// ---- Templates/GVLs/DPAD/Labels/Composition/LblCmpAC.TcGVL
{region '#Template'}
	{attribute 'Version' := '0.0.1.0'}
	{attribute 'Tags' := '"LCID": "1031", "Text": "GVL, AC, DPAD, Plants, ObjectName, Description"'}
	{attribute 'Tags' := '"LCID": "1033", "Text": "GVL, AC, DPAD, Plants, ObjectName, Description"'}
	{attribute 'Description' := '"LCID": "1031", "Text": "AC Labels Kompensation"'}
	{attribute 'Description' := '"LCID": "1033", "Text": "AC labels compensation"'}
{endregion}

{attribute 'qualified_only'}
VAR_GLOBAL
///////////////////////
//	Aggregates\Cooler	
	Cooler_TFl							:FB_BA_Label	:= LblAggregates.TemperatureFlow;	
	Cooler_TRt							:FB_BA_Label	:= LblAggregates.TemperatureReturnFlow;	

	Cooler_HSuACtrl_Ctrl				:FB_BA_Label	:= LblFunctions.LoopObject; 
	Cooler_HSuACtrl_Dehumf				:FB_BA_Label	:= LblControl.OperationalMessageDehumidification;	

	Cooler_TSuACtrl						:FB_BA_Label	:= LblControl.SupplyAirTemperatureControl;
	Cooler_TSuACtrl_Ctrl				:FB_BA_Label	:= LblFunctions.LoopObject; 

	Cooler_Vlv							:FB_BA_Label	:= LblAggregates.Valve;
	Cooler_Pu							:FB_BA_Label	:= LblAggregates.Pump;

//	Aggregates\ERC
	ERC_DiffPrssSwi						:FB_BA_Label	:= LblAggregates.PressureDifferential;												 										 
	ERC_IcePrtcRamp						:FB_BA_Label	:= LblControl.EnergyRecoveryDeicingRamp;
	ERC_Motor							:FB_BA_Label	:= LblAggregates.HeatRecovery;
	ERC_TExhACtrl						:FB_BA_Label	:= LblControl.ExhaustAirTemperatureControl;
	ERC_TSuACtrl						:FB_BA_Label	:= LblControl.SupplyAirTemperatureControl;
	ERC_TSuACtrl_Ctrl					:FB_BA_Label	:= LblFunctions.LoopObject; 

	ERC_DiffPrssSensor					:FB_BA_Label	:= LblAggregates.PressureDifferential;	
	ERC_Damping							:FB_BA_Label	:= LblAggregates.PressureDifferential;
	ERC_IcePrtcDiffPrssCtrl				:FB_BA_Label	:= LblControl.ExhaustAirTemperatureControl;
	ERC_Dmp								:FB_BA_Label	:= LblAggregates.VentilationDamperSupplyAir;	
	ERC_ByDmp							:FB_BA_Label	:= LblAggregates.VentilationDamperBypassAir;

//	Aggregates\Humidifier
	Humf_SuACtrl_Ctrl					:FB_BA_Label	:= LblFunctions.LoopObject; 
		
//	Aggregates\MixedAir
	Mix_TSuACtrl						:FB_BA_Label	:= LblControl.SupplyAirTemperatureControl;
	Mix_TSuACtrl_Ctrl					:FB_BA_Label	:= LblFunctions.LoopObject; 
	Mix_StartUpRamp						:FB_BA_Label	:= LblControl.MixedAirStartUpRamp;
	Mix_DmpMixA							:FB_BA_Label	:= LblAggregates.VentilationDamperMixAir;	
	Mix_DmpOuA							:FB_BA_Label	:= LblAggregates.VentilationDamperOutsideAir;	
	Mix_DmpExhA							:FB_BA_Label	:= LblAggregates.VentilationDamperExhaustAir;	

//	Aggregates\pre-heater
	PreHtr_TFl							:FB_BA_Label	:= LblAggregates.TemperatureFlow;	
	PreHtr_TRt							:FB_BA_Label	:= LblAggregates.TemperatureReturnFlow;	
	PreHtr_TSuACtrl						:FB_BA_Label	:= LblControl.SupplyAirTemperatureControl;
	PreHtr_TSuACtrl_Ctrl				:FB_BA_Label	:= LblFunctions.LoopObject; 
	PreHtr_TFrost						:FB_BA_Label	:= LblControl.TemperatureFrost;	
	PreHtr_TFrostPrtcCtrlAir			:FB_BA_Label	:= LblControl.FrostProtectionControl;
	PreHtr_FrostThermostat				:FB_BA_Label	:= LblAggregates.FrostProtectionMonitor;												 										 
	PreHtr_FrostThermostat_Input		:FB_BA_Label	:= LblFunctions.DangerAlarm;
	PreHtr_Vlv							:FB_BA_Label	:= LblAggregates.Valve;
	PreHtr_Pu							:FB_BA_Label	:= LblAggregates.Pump;		
	PreHtr_TRtCtrl						:FB_BA_Label	:= LblControl.ReturnWaterControl;
	PreHtr_TRtCtrl_SpTRtW				:FB_BA_Label	:= LblFunctions.Setpoint;
	PreHtr_TRtCtrl_PreRinseDelay		:FB_BA_Label	:= LblControl.DelayOn;
	PreHtr_TRtCtrl_PreRinseDelay_TiDly	:FB_BA_Label	:= LblControl.PreRinseDuration;
	PreHtr_TRtCtrl_PreRinseDst			:FB_BA_Label	:= LblControl.DisturbancePreRinse;	 								 
	PreHtr_TRtCtrl_PreRinseSp			:FB_BA_Label	:= LblControl.CalculationPreRinseSetpoint;			
	PreHtr_TRtCtrl_Ctrl					:FB_BA_Label	:= LblFunctions.LoopObject; 		
	
	PreHtr_ProcessPreRinse				:FB_BA_LabelProcess	:= LblControl.ProcPreRinse;

//	Aggregates\re-heater
	ReHtr_TFl							:FB_BA_Label	:= LblAggregates.TemperatureFlow;	
	ReHtr_TRt							:FB_BA_Label	:= LblAggregates.TemperatureReturnFlow;	
	ReHtr_TSuACtrl						:FB_BA_Label	:= LblControl.SupplyAirTemperatureControl;
	ReHtr_TSuACtrl_Ctrl					:FB_BA_Label	:= LblFunctions.LoopObject; 
	ReHtr_Vlv							:FB_BA_Label	:= LblAggregates.Valve;
	ReHtr_Pu							:FB_BA_Label	:= LblAggregates.Pump;		
		
///////////////////////
//	General
	General_OpModMan					:FB_BA_Label	:= LblControl.OperationModeSelection;							
	General_Sched						:FB_BA_Label	:= LblFunctions.Scheduler;							
	General_OpModPr						:FB_BA_Label	:= LblControl.PresentOperationMode;		
	
//	Summer night cooling
	General_SumNgtCol_WthTLoLmt			:FB_BA_Label	:= LblControl.OutsideTemperatureLowLimit;			
	General_SumNgtCol_RmTHys			:FB_BA_Label	:= LblControl.HysteresisRoomTemperature;			
	General_SumNgtCol_SwiOnDiffT		:FB_BA_Label	:= LblControl.OnValueDifferenceOutsideInsightTemperature;			
	General_SumNgtCol_SwiOffDiffT		:FB_BA_Label	:= LblControl.OffValueDifferenceOutsideInsightTemperature;			
	General_SumNgtCol_Q					:FB_BA_Label	:= LblFunctions.OperationalMessage;												 
	General_SumNgtCol_Sched				:FB_BA_Label	:= LblFunctions.Scheduler;		
///////////////////////
//	Setpoint\Temperature
	SpTRm_X1							:FB_BA_Label	:= LblControl.X01;	
	SpTRm_X2							:FB_BA_Label	:= LblControl.X02;	
	SpTRm_X3							:FB_BA_Label	:= LblControl.X03;	
	SpTRm_X4							:FB_BA_Label	:= LblControl.X04;	
	
	SpTRm_Y1							:FB_BA_Label	:= LblControl.Y01;
	SpTRm_Y2_3							:FB_BA_Label	:= LblControl.Y02_03;
	SpTRm_Y4							:FB_BA_Label	:= LblControl.Y03;
	SpTRm_Sp							:FB_BA_Label	:= LblFunctions.SetpointCalculated;
	
	SpTRm_SpColX1						:FB_BA_Label	:= LblControl.SummerCompensationX1;	
	SpTRm_SpColX2						:FB_BA_Label	:= LblControl.SummerCompensationX2;	
	SpTRm_SpColY1						:FB_BA_Label	:= LblControl.SummerCompensationY1;	
	SpTRm_SpColY2						:FB_BA_Label	:= LblControl.SummerCompensationY2;	
	SpTRm_SpColYMin						:FB_BA_Label	:= LblControl.SummerCompensationYmin;
	SpTRm_SpColYMax						:FB_BA_Label	:= LblControl.SummerCompensationYmax;	
	SpTRm_SpCol							:FB_BA_Label	:= LblControl.SummerCompensationSp;	
	
	SpTRm_SpHtgX1						:FB_BA_Label	:= LblControl.WinterCompensationX1;	
	SpTRm_SpHtgX2						:FB_BA_Label	:= LblControl.WinterCompensationX2;	
	SpTRm_SpHtgY1						:FB_BA_Label	:= LblControl.WinterCompensationY1;	
	SpTRm_SpHtgY2						:FB_BA_Label	:= LblControl.WinterCompensationY2;	
	SpTRm_SpHtgYMin						:FB_BA_Label	:= LblControl.WinterCompensationYmin;
	SpTRm_SpHtgYMax						:FB_BA_Label	:= LblControl.WinterCompensationYmax;		
	SpTRm_SpHtg							:FB_BA_Label	:= LblControl.WinterCompensationSp;	
	
	SpTSuA_SelSpErc						:FB_BA_Label	:= LblControl.OperationModeSelection;							
	SpTSuA_SpErc						:FB_BA_Label	:= LblFunctions.SetpointCalculated;	

	TCasCtrl_SpHtg						:FB_BA_Label	:= LblControl.SuppyAirTempSetpointHeaterCalc;			
	TCasCtrl_SpCol						:FB_BA_Label	:= LblControl.SuppyAirTempSetpointCoolerCalc;			
	TCasCtrl_SpErc						:FB_BA_Label	:= LblControl.SuppyAirTempSetpointERCCalc;			
	TCasCtrl_Ctrl						:FB_BA_Label	:= LblFunctions.LoopObjectCascadeSupplyAirTemperature; 			
	TCasCtrl_SelSpErc					:FB_BA_Label	:= LblControl.OperationModeSelection;							
//	Setpoint\Humidity
	HumCasCtrl_Ctrl						:FB_BA_Label	:= LblFunctions.LoopObjectCascadeSupplyAirHumidity; 	
	SpHum_SpH							:FB_BA_Label	:= LblControl.SetpointRelHumidity;			
	SpHum_SpX							:FB_BA_Label	:= LblControl.SetpointCalculatedAbsHumidity;
	SpHum_SpHHumf						:FB_BA_Label	:= LblControl.SetpointRelHumidityHumidification;			
	SpHum_SpHDehumf						:FB_BA_Label	:= LblControl.SetpointRelHumidityDehumidification;			
	SpHum_SpXHumf						:FB_BA_Label	:= LblControl.SetpointCalculatedAbsHumidityHumidification;	
	SpHum_SpXDehumf						:FB_BA_Label	:= LblControl.SetpointCalculatedAbsHumidityDehumidification;


//	Sonderlösung - eventuelle Überarbeitung
	PlantControlStatus   	:FB_BA_Label2x :=(iAggregate:=LblControl.PlantControl,		iFunction:=LblFunctions.Status);
	TSequenceControlStatus  :FB_BA_Label2x :=(iAggregate:=LblControl.TSequenceControl,	iFunction:=LblFunctions.Status);		

//	AHU	
	AHU_TOuA						:FB_BA_Label	:= LblAggregates.TemperatureOutside;	
	AHU_TExhA						:FB_BA_Label	:= LblAggregates.TemperatureExhaustAir;	
	AHU_TSuA						:FB_BA_Label	:= LblAggregates.TemperatureSupplyAir;	
	AHU_TExtA						:FB_BA_Label	:= LblAggregates.TemperatureExtractAir;	
	AHU_TRm							:FB_BA_Label	:= LblAggregates.TemperatureRoomAir;	
	AHU_DiffPrssOuAFilt				:FB_BA_Label	:= LblAggregates.PressureDifferentialOutsideAirFilter;	
	AHU_FiltOuAMonit				:FB_BA_Label	:= LblAggregates.AirFilterOutsideAir;
	AHU_DiffPrssExtAFilt			:FB_BA_Label	:= LblAggregates.PressureDifferentialExtractAirFilter;	
	AHU_FiltExtAMonit				:FB_BA_Label	:= LblAggregates.AirFilterExtractAir;
	AHU_SumNgtCol					:FB_BA_Label	:= LblControl.SummerNightCooling;
	AHU_OpMod						:FB_BA_Label	:= LblControl.OperationMode;
	AHU_OuADmp						:FB_BA_Label	:= LblAggregates.VentilationDamperOutsideAir;
	AHU_SuAPrss						:FB_BA_Label	:= LblAggregates.PressureSupplyAir;	
	AHU_SuADiffPrss					:FB_BA_Label	:= LblAggregates.PressureDifferentialSupplyAirFan;	
	AHU_SuAFan						:FB_BA_Label	:= LblAggregates.FanSupplyAir;
	AHU_SuADiffPrssMonit			:FB_BA_Label	:= LblControl.DifferencePressureMonitoringSupplyAirFan;
	AHU_ExhADmp						:FB_BA_Label	:= LblAggregates.VentilationDamperExhaustAir;
	AHU_ExtAPrss					:FB_BA_Label	:= LblAggregates.PressureExtractAir;	
	AHU_ExtADiffPrss				:FB_BA_Label	:= LblAggregates.PressureDifferentialExtractAirFan;	
	AHU_ExtAFan						:FB_BA_Label	:= LblAggregates.FanExtractAir;
	AHU_ExtADiffPrssMonit			:FB_BA_Label	:= LblControl.DifferencePressureMonitoringExtractAirFan;
	AHU_SpTRm						:FB_BA_Label	:= LblControl.SetpointCalculation;
	AHU_TCasCtrl					:FB_BA_Label	:= LblControl.CascadeSupplyAirControl;
	AHU_TSeqLink					:FB_BA_Label2x	:= TSequenceControlStatus;
	AHU_PreHtr						:FB_BA_Label	:= LblControl.PreHeater;
	AHU_Erc							:FB_BA_Label	:= LblControl.EnergyRecovery;
	AHU_Col							:FB_BA_Label	:= LblControl.Cooler;
	AHU_PlantCtrl					:FB_BA_Label2x	:= PlantControlStatus;	



	
END_VAR

// ---- Templates/GVLs/DPAD/Labels/Composition/LblCmpGeneral.TcGVL
{region '#Template'}
	{attribute 'Version' := '0.0.1.0'}
	{attribute 'Tags' := '"LCID": "1031", "Text": "GVL, General, DPAD, Plants, ObjectName, Description"'}
	{attribute 'Tags' := '"LCID": "1033", "Text": "GVL, General, DPAD, Plants, ObjectName, Description"'}
	{attribute 'Description' := '"LCID": "1031", "Text": "Allgemein Labels Kompensation"'}
	{attribute 'Description' := '"LCID": "1033", "Text": "General labels compensation"'}
{endregion}

{attribute 'qualified_only'}
VAR_GLOBAL
	BuildingAlarms_FireAlert						: FB_BA_Label := LblControl.FireAlert;
	BuildingAlarms_Bgly								: FB_BA_Label := LblControl.Burglary;
	BuildingAlarms_CentSwiOff						: FB_BA_Label := LblControl.CentralSwitchOff;
                                  				
	BuildingMode_OpModMan							: FB_BA_Label := LblControl.BuildingModeManual;
	BuildingMode_OpModPr							: FB_BA_Label := LblControl.BuildingModeActual;
	BuildingMode_Sched								: FB_BA_Label := LblControl.BuildingModeSched;
                                  				
	BuildingGlobal_BuildAlm							: FB_BA_Label := LblControl.BuildingAlarms;
	BuildingGlobal_BuildMode						: FB_BA_Label := LblControl.BuildingMode;
	
	ControlCabinet_Fuse								: FB_BA_Label := LblControl.Fuse;	
	ControlCabinet_Fuse_Input						: FB_BA_Label := LblFunctions.Fault;	
	ControlCabinet_LampFault						: FB_BA_Label := LblControl.EventIndicationLamp;			
	ControlCabinet_LampFault_Cmd					: FB_BA_Label := LblFunctions.SwitchingCommand;			
	ControlCabinet_AckButton 						: FB_BA_Label := LblControl.Acknowledge;	
	ControlCabinet_AckButton_Input					: FB_BA_Label := LblControl.ButtonLocalAcknowledgement;
	ControlCabinet_AckButton_Value					: FB_BA_Label := LblControl.ButtonRemoteAcknowledgement;
	ControlCabinet_RstHw							: FB_BA_Label := LblControl.AcknowledgeCommand;			
	ControlCabinet_RstHw_Cmd						: FB_BA_Label := LblFunctions.SwitchingCommand;	
	
	EvtGroups_LifeSafety							: FB_BA_Label := LblControl.EvtCategoryLifeSafty;									  
	EvtGroups_AlarmTechnical						: FB_BA_Label := LblControl.EvtCategoryAlarmTechnical;									  
	EvtGroups_Disturbance							: FB_BA_Label := LblControl.EvtCategoryDisturbance;									  
	EvtGroups_Maintenance							: FB_BA_Label := LblControl.EvtCategoryMaintenance;									  
	EvtGroups_Notification							: FB_BA_Label := LblControl.EvtCategoryNotification;									  
	EvtGroups_Other									: FB_BA_Label := LblControl.EvtCategoryOther;									  
	
	Settings_WthParam								: FB_BA_Label := LblControl.WeatherParameters;	
	
	WthParam_SpFrstProtec							: FB_BA_Label := LblControl.SetpointFrostProtection;
	WthParam_TWthLowLimitVal						: FB_BA_Label := LblControl.SetpointMinimumOutsideTemperature;
	WthParam_TWthLowLimit							: FB_BA_Label := LblControl.OperationalMessageTemperatureWeatherLowLimit;	
	WthParam_TWthDamped								: FB_BA_Label := LblControl.MeanDamped;
	WthParam_TWthDampedLowLimit						: FB_BA_Label := LblControl.OperationalMessageTemperatureWeatherDampedLowLimit;	
END_VAR

// ---- Templates/GVLs/DPAD/Labels/Composition/LblCmpRoomAutomation.TcGVL
{region '#Template'}
	{attribute 'Version' := '0.0.1.0'}
	{attribute 'Tags' := '"LCID": "1031", "Text": "GVL, Room automation, DPAD, Plants, ObjectName, Description"'}
	{attribute 'Tags' := '"LCID": "1033", "Text": "GVL, Room automation, DPAD, Plants, ObjectName, Description"'}
	{attribute 'Description' := '"LCID": "1031", "Text": "Raum Automation Labels Kompensation"'}
	{attribute 'Description' := '"LCID": "1033", "Text": "Room automation labels compensation"'}
{endregion}

{attribute 'qualified_only'}
VAR_GLOBAL
	BuildingEnergyLevel_EnergLvlMan					: FB_BA_Label := LblControl.BuildingEnergyLevelManual;
	BuildingEnergyLevel_EnergLvlPr					: FB_BA_Label := LblControl.BuildingEnergyLevelActual;
	BuildingEnergyLevel_Sched						: FB_BA_Label := LblControl.BuildingEnergyLevelSched;
    
	BuildingSpRmT_SumCpsn							: FB_BA_Label := LblControl.SummerCompensation;
	BuildingSpRmT_WinCpsn							: FB_BA_Label := LblControl.WinterCompensation;
	BuildingSpRmT_PrtcHtg							: FB_BA_Label := LblFunctions.SetpointProtectionHeating;
	BuildingSpRmT_EcoHtg							: FB_BA_Label := LblFunctions.SetpointEconomyHeating;
	BuildingSpRmT_PreCmfHtg							: FB_BA_Label := LblFunctions.SetpointPreComfortHeating;
	BuildingSpRmT_CmfHtg							: FB_BA_Label := LblFunctions.SetpointComfortHeating;
	BuildingSpRmT_PrtcCol							: FB_BA_Label := LblFunctions.SetpointProtectionCooling;
	BuildingSpRmT_EcoCol							: FB_BA_Label := LblFunctions.SetpointEconomyCooling;
	BuildingSpRmT_PreCmfCol							: FB_BA_Label := LblFunctions.SetpointPreComfortCooling;
	BuildingSpRmT_CmfCol							: FB_BA_Label := LblFunctions.SetpointComfortCooling;
	BuildingSpRmT_ShiftHtg							: FB_BA_Label := LblControl.SetpointShiftHeating;
	BuildingSpRmT_ShiftCol							: FB_BA_Label := LblControl.SetpointShiftCooling;
	
	BuildingSunprotection_SpIce						: FB_BA_Label := LblControl.SetpointIce;
	BuildingSunprotection_SunPrtcPosIntval			: FB_BA_Label := LblControl.SunProtectionInterval;
	BuildingSunprotection_DeiceTi					: FB_BA_Label := LblControl.DeiceTime;
	BuildingSunprotection_GlobalThAutoValOn			: FB_BA_Label := LblControl.GlobalThermoAutomaticValueOn;
	BuildingSunprotection_GlobalThAutoValOff		: FB_BA_Label := LblControl.GlobalThermoAutomaticValueOff;
	BuildingSunprotection_GlobalTwiLgtAutoValOn		: FB_BA_Label := LblControl.GlobalTwilightAutomaticValueOn;
	BuildingSunprotection_GlobalTwiLgtAutoValOff	: FB_BA_Label := LblControl.GlobalTwilightAutomaticValueOff;
	BuildingSunprotection_IceAlert					: FB_BA_Label := LblControl.IceAlert;
	BuildingSunprotection_GlobalThAutoRlse			: FB_BA_Label := LblControl.GlobalThermoAutomaticRelease;
	BuildingSunprotection_GlobalTwiLgtAutoRlse		: FB_BA_Label := LblControl.GlobalTwilightAutomaticRelease;
	BuildingSunprotection_GlobalResetManMode		: FB_BA_Label := LblControl.GlobalResetManMode;
	
	Facade_DlyStrmOn								: FB_BA_Label := LblControl.TimeDelayStormOn;
	Facade_DlyStrmOff								: FB_BA_Label := LblControl.TimeDelayStormOff;
	Facade_MntnEn									: FB_BA_Label := LblControl.MaintenanceEnable;                    		
	Facade_MntnPos									: FB_BA_Label := LblControl.MaintenancePosition;
	Facade_MntnAngl									: FB_BA_Label := LblControl.MaintenanceAngle;
	Facade_FcdThAutoEn								: FB_BA_Label := LblControl.FacadeThermoAutomaticEnable;
	Facade_FcdThAutoColPos							: FB_BA_Label := LblControl.FacadeThermoAutomaticCoolingPosition;
	Facade_FcdThAutoColAngl							: FB_BA_Label := LblControl.FacadeThermoAutomaticCoolingAngle;
	Facade_FcdTwiLgtAutoEn							: FB_BA_Label := LblControl.FacadeTwilightAutomaticEnable;
	Facade_SunPrtcValOn								: FB_BA_Label := LblControl.SunProtectionValueOn;
	Facade_SunPrtcValOff							: FB_BA_Label := LblControl.SunProtectionValueOff;
	Facade_SunPrtcDlyOn								: FB_BA_Label := LblControl.TimeDelaySunProtectionOn;
	Facade_SunPrtcDlyOff							: FB_BA_Label := LblControl.TimeDelaySunProtectionOff;
	Facade_FcdParkEn								: FB_BA_Label := LblControl.FacadeParkingEnable;
	Facade_FcdParkPos								: FB_BA_Label := LblControl.FacadeParkingPosition;
	Facade_FcdParkAngl								: FB_BA_Label := LblControl.FacadeParkingAngle;
	Facade_WndPrtcState								: FB_BA_Label := LblControl.WindProtectionState;
	Facade_SunPrtcState								: FB_BA_Label := LblControl.SunProtectionState;
    
	SunBld_LocInputPos								: FB_BA_Label := LblControl.SetpointSunblindPosition;
	SunBld_LocInputAngl								: FB_BA_Label := LblControl.SetpointSunblindAngle;
	SunBld_LocButtonStart							: FB_BA_Label := LblControl.CommandSunblindStart;
	SunBld_ActlPos									: FB_BA_Label := LblControl.FeedbackSunblindPosition;
	SunBld_ActlAngl									: FB_BA_Label := LblControl.FeedbackSunblindAngle;
	SunBld_ActlPrio									: FB_BA_Label := LblControl.FeedbackSunblindPrio;
	SunBld_ManSwi									: FB_BA_Label := LblControl.ButtonSunblind;
		
	HeatCoolAxisAnlg_RmTSen							: FB_BA_Label := LblAggregates.TemperatureRoomAir;
	HeatCoolAxisAnlg_RmTAdj							: FB_BA_Label := LblAggregates.RoomControlUnit;
	HeatCoolAxisAnlg_PrtcDetc						: FB_BA_Label := LblAggregates.PresenceSwitches;
	HeatCoolAxisAnlg_WdwCon							: FB_BA_Label := LblAggregates.WindowContact;
	HeatCoolAxisAnlg_VlvHtg							: FB_BA_Label :=(sObjName:='VEN',sDescr:='Heizventil');
 	HeatCoolAxisAnlg_VlvCol							: FB_BA_Label :=(sObjName:='VEN',sDescr:='Kuehlventil');
 	HeatCoolAxisAnlg_Ctrl							: FB_BA_Label := LblControl.RoomTemperatureControl;
 	HeatCoolAxisAnlg_Ctrl_CtrlHtg					: FB_BA_Label :=(sObjName:='LPH',sDescr:='Heizregler');
 	HeatCoolAxisAnlg_Ctrl_CtrlCol					: FB_BA_Label :=(sObjName:='LPC',sDescr:='Kuehlregler');
	HeatCoolAxisAnlg_DewPoint						: FB_BA_Label := LblAggregates.MonitorDewPoint;

	SunBldZone_SunBld								: FB_BA_Label := LblAggregates.Blind;
                                          	
//	RoomAutomation_RoomGeneral						: FB_BA_Label := LabelPlants.Room_automation;
	
	RoomGeneral_FcdEast								: FB_BA_Label := LblControl.Facade;
END_VAR

// ---- Templates/GVLs/DPAD/Texts/1031/TxtEvent_1031.TcGVL
{region '#Template'}
	{attribute 'Version' := '1.0.0.0'}
	{attribute 'Tags' := '"LCID": "1031", "Text": "GVL, Property, Event, Event Message Text, Active Text, Inactive Text, State Text"'}
	{attribute 'Tags' := '"LCID": "1033", "Text": "GVL, Property, Event, Event Message Text, Active Text, Inactive Text, State Text"'}
	{attribute 'Description' := '"LCID": "1031", "Text": "Textliste Properties Event Message Text, Active Text, Inactive Text, State Text"'}
	{attribute 'Description' := '"LCID": "1033", "Text": "Text list Properties Event Message Text, Active Text, Inactive Text, State Text"'}
{endregion}

{attribute 'global_init_slot' := '40510'}
VAR_GLOBAL
  txtEvent_No                                                :T_BA_StateText:='Nein';
  txtEvent_Yes                                               :T_BA_StateText:='Ja';
  txtEvent_Auto                                              :T_BA_StateText:='Automatik';
  txtEvent_Manual                                            :T_BA_StateText:='Hand';
  txtEvent_Off                                               :T_BA_StateText:='Aus';
  txtEvent_On                                                :T_BA_StateText:='Ein';
  txtEvent_Opened                                            :T_BA_StateText:='Geöffnet';
  txtEvent_Closed                                            :T_BA_StateText:='Geschlossen';
  txtEvent_Open                                              :T_BA_StateText:='Auf';
  txtEvent_Close                                             :T_BA_StateText:='Zu';
  txtEvent_Step1                                             :T_BA_StateText:='Stufe 1 ';
  txtEvent_Step2                                             :T_BA_StateText:='Stufe 2';
  txtEvent_Step3                                             :T_BA_StateText:='Stufe 3';
  txtEvent_Released                                          :T_BA_StateText:='Freigegeben';
  txtEvent_Inactive                                          :T_BA_StateText:='Inaktiv';
  txtEvent_Active                                            :T_BA_StateText:='Aktiv';
  txtEvent_Normal                                            :T_BA_StateText:='Normal';
  txtEvent_Offnormal                                         :T_BA_StateText:='Unnormal';
  txtEvent_Alert                                             :T_BA_StateText:='Alarm';
  txtEvent_Disturb                                           :T_BA_StateText:='Störung';
  txtEvent_Error                                             :T_BA_StateText:='Fehler ';
  txtEvent_Triggered                                         :T_BA_StateText:='Ausgelöst';
  txtEvent_Maintenace                                        :T_BA_StateText:='Wartung';
  txtEvent_Exceeded                                          :T_BA_StateText:='Überschritten';
  txtEvent_Monitoring                                        :T_BA_StateText:='Überwachung';
  txtEvent_Protection                                        :T_BA_StateText:='Schutzbetrieb';
  txtEvent_Economy                                           :T_BA_StateText:='Economy';
  txtEvent_PreComfort                                        :T_BA_StateText:='Pre-Comfort';
  txtEvent_Comfort                                           :T_BA_StateText:='Comfort';
  txtEvent_Reached                                           :T_BA_StateText:='erreicht';
  txtEvent_NotReached                                        :T_BA_StateText:='nicht erreicht';
  txtEvent_None                                              :T_BA_StateText:='""';
  txtEvent_EmergencyStop                                     :T_BA_StateText:='Notaus';
  txtEvent_Frost                                             :T_BA_StateText:='Frost';
  txtEvent_SmokeExtraction_P                                 :T_BA_StateText:='Entrauchung mit Zu- und Abluft';
  txtEvent_SmokeExtractionSupplyAir                          :T_BA_StateText:='Entrauchung Zuluft';
  txtEvent_SmokeExtractionExtractAir                         :T_BA_StateText:='Entrauchung Abluft';
  txtEvent_CoolDownProtection                                :T_BA_StateText:='Auskühlschutz';
  txtEvent_OverHeatingProtection                             :T_BA_StateText:='Überhitzungsschutz';
  txtEvent_Fire                                              :T_BA_StateText:='Brandalarm';
  txtEvent_NightCooling                                      :T_BA_StateText:='Nachtkühlung';
  txtEvent_ForcedVentilation                                 :T_BA_StateText:='Zwangsbelüftung';
  txtEvent_CentralSwitchOff                                  :T_BA_StateText:='Zentralaus';
  txtEvent_Locked                                            :T_BA_StateText:='verriegelt';
  txtEvent_Contaminated                                      :T_BA_StateText:='verschmutzt';
  txtEvent_Stop                                              :T_BA_StateText:='Stop';
  txtEvent_Critical                                          :T_BA_StateText:='kritisch';
  txtEvent_UnCiritical                                       :T_BA_StateText:='unkritisch';
  txtEvent_Average                                           :T_BA_StateText:='Mittelwert';
  txtEvent_HeatCool                                          :T_BA_StateText:='Heiz/Kühl';
  txtEvent_AverageHeatCool                                   :T_BA_StateText:='Mittelwert Heizen/Kühlen';
  txtEvent_Direction                                         :T_BA_StateText:='Wirksinn';
  txtEvent_Default                                           :T_BA_StateText:='Standard';
  txtEvent_Cleaning                                          :T_BA_StateText:='Gebaeudereinigung';
  txtEvent_Nightwatch                                        :T_BA_StateText:='Nachtwaechter';
  txtEvent_SupplyAirTControlReheater                         :T_BA_StateText:='Zulufttemperaturregelung Nacherhitzer';
  txtEvent_SupplyAirTControlPeheater                         :T_BA_StateText:='Zulufttemperaturregelung Vorerhitzer';
  txtEvent_SupplyAirTControlERC                              :T_BA_StateText:='Zulufttemperaturregelung WRG';
  txtEvent_SupplyAirTControlMix                              :T_BA_StateText:='Zulufttemperaturregelung Mischluft';
  txtEvent_SupplyAirTControlCooler                           :T_BA_StateText:='Zulufttemperaturregelung Kühler';
  txtEvent_SupplyAirXControlCooler                           :T_BA_StateText:='Zuluftfeuchtereglung Kühler';
  txtEvent_SupplyAirXControlHumf                             :T_BA_StateText:='Zuluftfeuchtereglung Befeuchter';
END_VAR

// ---- Templates/GVLs/DPAD/Texts/1031/TxtTrade_1031.TcGVL
{region '#Template'}
	{attribute 'Version' := '1.0.0.0'}
	{attribute 'Tags' := '"LCID": "1031", "Text": "GVL, DPAD, Trades, ObjectName, Description"'}
	{attribute 'Tags' := '"LCID": "1033", "Text": "GVL, DPAD, Trades, ObjectName, Description"'}
	{attribute 'Description' := '"LCID": "1031", "Text": "Textliste Gewerke"'}
	{attribute 'Description' := '"LCID": "1033", "Text": "Text list trades"'}
{endregion}

{attribute 'global_init_slot' := '40510'}
VAR_GLOBAL
  TxtTrade_Doors_gates_windows_sun_protection_sObjectName                :T_BA_StateText:='TTF';
  TxtTrade_Doors_gates_windows_sun_protection_sDescription                :T_BA_StateText:='Türen, Tore, Fenster, Sonnenschutz';
  TxtTrade_Sewage_water_and_gas_plants_sObjectName                       :T_BA_StateText:='GWA';
  TxtTrade_Sewage_water_and_gas_plants_sDescription                       :T_BA_StateText:='Abwasser-, Wasser-, Gasanlagen';
  TxtTrade_Heat_supply_systems_sObjectName                               :T_BA_StateText:='HZG';
  TxtTrade_Heat_supply_systems_sDescription                               :T_BA_StateText:='Wärmeversorgungsanlagen';
  TxtTrade_Air_conditioning_sObjectName                                  :T_BA_StateText:='LTA';
  TxtTrade_Air_conditioning_sDescription                                  :T_BA_StateText:='Lufttechnische Anlagen';
  TxtTrade_Refrigeration_systems_sObjectName                             :T_BA_StateText:='KAE';
  TxtTrade_Refrigeration_systems_sDescription                             :T_BA_StateText:='Kälteanlagen';
  TxtTrade_High_voltage_systems_sObjectName                              :T_BA_StateText:='ELT';
  TxtTrade_High_voltage_systems_sDescription                              :T_BA_StateText:='Starkstromanlagen';
  TxtTrade_Telecommunication_and_information_technology_sObjectName      :T_BA_StateText:='FIA';
  TxtTrade_Telecommunication_and_information_technology_sDescription      :T_BA_StateText:='Fernm.- und informationstech. Anlagen';
  TxtTrade_Hazard_detection_and_alarm_systems_sObjectName                :T_BA_StateText:='GMA';
  TxtTrade_Hazard_detection_and_alarm_systems_sDescription                :T_BA_StateText:='Gefahrenmelde- und Alarmanlagen';
  TxtTrade_Conveyors_sObjectName                                         :T_BA_StateText:='FTA';
  TxtTrade_Conveyors_sDescription                                         :T_BA_StateText:='Förderanlagen';
  TxtTrade_Kitchen_technology_systems_sObjectName                        :T_BA_StateText:='KTA';
  TxtTrade_Kitchen_technology_systems_sDescription                        :T_BA_StateText:='Küchentechnische Anlagen';
  TxtTrade_Laundry_and_cleaning_systems_sObjectName                      :T_BA_StateText:='WAR';
  TxtTrade_Laundry_and_cleaning_systems_sDescription                      :T_BA_StateText:='Wäscherei- und Reinigungsanlagen';
  TxtTrade_Media_supply_systems_sObjectName                              :T_BA_StateText:='MVA';
  TxtTrade_Media_supply_systems_sDescription                              :T_BA_StateText:='Medienversorgungsanlagen';
  TxtTrade_Medical_and_laboratory_equipment_sObjectName                  :T_BA_StateText:='MED';
  TxtTrade_Medical_and_laboratory_equipment_sDescription                  :T_BA_StateText:='Medizin- und labortechnische Anlagen';
  TxtTrade_Fire_extinguishing_systems_sObjectName                        :T_BA_StateText:='FLA';
  TxtTrade_Fire_extinguishing_systems_sDescription                        :T_BA_StateText:='Feuerlöschanlagen';
  TxtTrade_Bathing_facilities_sObjectName                                :T_BA_StateText:='BTA';
  TxtTrade_Bathing_facilities_sDescription                                :T_BA_StateText:='Badetechnische Anlagen';
  TxtTrade_Process_heating_cooling_and_air_systems_sObjectName           :T_BA_StateText:='PRO';
  TxtTrade_Process_heating_cooling_and_air_systems_sDescription           :T_BA_StateText:='Prozesswärme-, -kälte- und -luftanlagen';
  TxtTrade_Waste_disposal_facilities_sObjectName                         :T_BA_StateText:='ENT';
  TxtTrade_Waste_disposal_facilities_sDescription                         :T_BA_StateText:='Entsorgungsanlagen';
  TxtTrade_Building_automation_and_control_systems_general_sObjectName   :T_BA_StateText:='GAS';
  TxtTrade_Building_automation_and_control_systems_general_sDescription   :T_BA_StateText:='Gebäudeautomation allgemein';
  TxtTrade_Automation_focal_point_information_focal_point_sObjectName    :T_BA_StateText:='ASP';
  TxtTrade_Automation_focal_point_information_focal_point_sDescription    :T_BA_StateText:='Automationsschwerpunkt';
  TxtTrade_Room_automation_sObjectName                                   :T_BA_StateText:='RAU';
  TxtTrade_Room_automation_sDescription                                   :T_BA_StateText:='Raumautomation';
  TxtTrade_Outdoor_devices_sObjectName                                   :T_BA_StateText:='AUG';
  TxtTrade_Outdoor_devices_sDescription                                   :T_BA_StateText:='Außengeräte';
END_VAR

// ---- Templates/GVLs/DPAD/Texts/TextPlants.TcGVL
{region '#Template'}
	{attribute 'Version' := '0.0.1.0'}
	{attribute 'Tags' := '"LCID": "1031", "Text": "GVL, DPAD, Plants, ObjectName, Description"'}
	{attribute 'Tags' := '"LCID": "1033", "Text": "GVL, DPAD, Plants, ObjectName, Description"'}
	{attribute 'Description' := '"LCID": "1031", "Text": "Textliste Anlagen"'}
	{attribute 'Description' := '"LCID": "1033", "Text": "Text list plants"'}
{endregion}

{attribute 'qualified_only'}
{attribute 'global_init_slot' := '40510'}
// erstellt am :19.05.2021 -- 10:49:48 Liste Anlagenbezeichnungen nach VDI 3814
VAR_GLOBAL
  Facade_sObjectName                                            :T_BA_StateText:='FAS';
  Facade_sDescription                                            :T_BA_StateText:='Fassade';
  Natural_smoke_extraction_sObjectName                          :T_BA_StateText:='NRA';
  Natural_smoke_extraction_sDescription                          :T_BA_StateText:='Natürlicher Rauchabzug';
  Doors_gates_sluices_sObjectName                               :T_BA_StateText:='TUE';
  Doors_gates_sluices_sDescription                               :T_BA_StateText:='Türen, Tore, Schleusen';
  Smoke_and_heat_extraction_system_sObjectName                  :T_BA_StateText:='RWA';
  Smoke_and_heat_extraction_system_sDescription                  :T_BA_StateText:='Rauch- und Wärmeabzugsanlage';
  Sunlight_protection_sObjectName                               :T_BA_StateText:='SON';
  Sunlight_protection_sDescription                               :T_BA_StateText:='Sonnenschutzanlage';
// 411 Abwasseranlagen
  Separator_facility_sObjectName                                :T_BA_StateText:='ABS';
  Separator_facility_sDescription                                :T_BA_StateText:='Abscheideranlage';
  Lifting_system_sObjectName                                    :T_BA_StateText:='HBA';
  Lifting_system_sDescription                                    :T_BA_StateText:='Hebeanlage';
  Neutralisation_plant_sObjectName                              :T_BA_StateText:='NEU';
  Neutralisation_plant_sDescription                              :T_BA_StateText:='Neutralisationsanlage';
// 412 Wasseranlagen
  Trace_heating_sObjectName                                     :T_BA_StateText:='BGH';
  Trace_heating_sDescription                                     :T_BA_StateText:='Begleitheizung';
  Process_water_sObjectName                                     :T_BA_StateText:='BTW';
  Process_water_sDescription                                     :T_BA_StateText:='Betriebswasser';
  Well_water_sObjectName                                        :T_BA_StateText:='BWA';
  Well_water_sDescription                                        :T_BA_StateText:='Brunnenwasser';
  Dispensing_installation_sObjectName                           :T_BA_StateText:='DOS';
  Dispensing_installation_sDescription                           :T_BA_StateText:='Dosieranlage';
  Pressure_booster_system_sObjectName                           :T_BA_StateText:='DEA';
  Pressure_booster_system_sDescription                           :T_BA_StateText:='Druckerhöhungsanlage';
  Softening_unit_sObjectName                                    :T_BA_StateText:='EHA';
  Softening_unit_sDescription                                    :T_BA_StateText:='Enthärtungsanlage';
// Trinkwasser
  Drinking_water_heating_system_sObjectName                     :T_BA_StateText:='TWE';
  Drinking_water_heating_system_sDescription                     :T_BA_StateText:='Trinkwassererwärmungsanlage';
  Reverse_osmosis_system_sObjectName                            :T_BA_StateText:='UKO';
  Reverse_osmosis_system_sDescription                            :T_BA_StateText:='Umkehrosmoseanlage';
  Desalination_plant_sObjectName                                :T_BA_StateText:='VEA';
  Desalination_plant_sDescription                                :T_BA_StateText:='Vollentsalzungsanlage';
// 421 Wärmeerzeugungsanlagen
  BHKW_sObjectName                                              :T_BA_StateText:='BHK';
  BHKW_sDescription                                              :T_BA_StateText:='BHKW';
  Electric_heating_sObjectName                                  :T_BA_StateText:='EHZ';
  Electric_heating_sDescription                                  :T_BA_StateText:='Elektroheizung';
  District_heating_transfer_sObjectName                         :T_BA_StateText:='FWÜ';
  District_heating_transfer_sDescription                         :T_BA_StateText:='Fernwärmeübergabe';
// Geothermieanlage
  Boiler_sObjectName                                            :T_BA_StateText:='KES';
  Boiler_sDescription                                            :T_BA_StateText:='Kessel';
  Clean_steam_generation_sObjectName                            :T_BA_StateText:='RDE';
  Clean_steam_generation_sDescription                            :T_BA_StateText:='Reindampferzeugung';
  Solar_power_system_sObjectName                                :T_BA_StateText:='SOL';
  Solar_power_system_sDescription                                :T_BA_StateText:='Solaranlage';
  Heating_pump_sObjectName                                      :T_BA_StateText:='WPU';
  Heating_pump_sDescription                                      :T_BA_StateText:='Wärmepumpe';
// 422 Wärmeverteilnetze
  Pressure_maintenance_sObjectName                              :T_BA_StateText:='DHG';
  Pressure_maintenance_sDescription                              :T_BA_StateText:='Druckhaltung';
  Heating_circuit_sObjectName                                   :T_BA_StateText:='HZK';
  Heating_circuit_sDescription                                   :T_BA_StateText:='Heizkreis';
  Heating_sObjectName                                           :T_BA_StateText:='HZG';
  Heating_sDescription                                           :T_BA_StateText:='Heizung (allgemein)';
  Back_feed_system_sObjectName                                  :T_BA_StateText:='NSA';
  Back_feed_system_sDescription                                  :T_BA_StateText:='Nachspeiseanlage';
  Buffer_sObjectName                                            :T_BA_StateText:='PFS';
  Buffer_sDescription                                            :T_BA_StateText:='Pufferspeicher';
  Heat_distribution_network_sObjectName                         :T_BA_StateText:='WVN';
  Heat_distribution_network_sDescription                         :T_BA_StateText:='Wärmeverteilnetz';
  Heat_exchanger_sObjectName                                    :T_BA_StateText:='WTR';
  Heat_exchanger_sDescription                                    :T_BA_StateText:='Wärmeüberträger';
// 423 Raumheizflächen
  Concrete_core_activation_sObjectName                          :T_BA_StateText:='BKA';
  Concrete_core_activation_sDescription                          :T_BA_StateText:='Betonkernaktivierung';
  Overhead_heating_sObjectName                                  :T_BA_StateText:='DHZ';
  Overhead_heating_sDescription                                  :T_BA_StateText:='Deckenheizung';
  Ceiling_radiator_panels_sObjectName                           :T_BA_StateText:='DSP';
  Ceiling_radiator_panels_sDescription                           :T_BA_StateText:='Deckenstrahlplatten';
  Facade_heating_sObjectName                                    :T_BA_StateText:='FAH';
  Facade_heating_sDescription                                    :T_BA_StateText:='Fassadenheizung';
  Panel_heating_sObjectName                                     :T_BA_StateText:='FLH';
  Panel_heating_sDescription                                     :T_BA_StateText:='Flächenheizung';
  Underfloor_heating_sObjectName                                :T_BA_StateText:='FBH';
  Underfloor_heating_sDescription                                :T_BA_StateText:='Fußbodenheizung';
  Heated_chilled_ceiling_sObjectName                            :T_BA_StateText:='HKD';
  Heated_chilled_ceiling_sDescription                            :T_BA_StateText:='Heiz-/Kühldecke';
  Static_heating_sObjectName                                    :T_BA_StateText:='STH';
  Static_heating_sDescription                                    :T_BA_StateText:='Statische Heizung';
// 430 Lufttechnische Anlagen
  Extract_air_system_sObjectName                                :T_BA_StateText:='ABA';
  Extract_air_system_sDescription                                :T_BA_StateText:='Abluftanlage';
  Roof_air_heater_sObjectName                                   :T_BA_StateText:='DLH';
  Roof_air_heater_sDescription                                   :T_BA_StateText:='Deckenlufterhitzer';
  Circulatory_system_sObjectName                                :T_BA_StateText:='KVS';
  Circulatory_system_sDescription                                :T_BA_StateText:='Kreislaufverbundsystem';
  Air_processing_unit_sObjectName                               :T_BA_StateText:='LAZ';
  Air_processing_unit_sDescription                               :T_BA_StateText:='Luftaufbereitungszentrale';
  Mechanical_smoke_extraction_system_sObjectName                :T_BA_StateText:='MRA';
  Mechanical_smoke_extraction_system_sDescription                :T_BA_StateText:='Maschinelle Rauchabzugsanlage';
  Smoke_pressure_system_sObjectName                             :T_BA_StateText:='RDA';
  Smoke_pressure_system_sDescription                             :T_BA_StateText:='Rauchdruckanlage';
  Air_handling_unit_sObjectName                                 :T_BA_StateText:='RLT';
  Air_handling_unit_sDescription                                 :T_BA_StateText:='Raumlufttechnik (allgemein)';
  Partial_air_conditioning_system_sObjectName                   :T_BA_StateText:='TKA';
  Partial_air_conditioning_system_sDescription                   :T_BA_StateText:='Teilklimaanlage';
  Air_curtain_system_sObjectName                                :T_BA_StateText:='TLS';
  Air_curtain_system_sDescription                                :T_BA_StateText:='Türluftschleieranlage';
  Recirculating_air_system_sObjectName                          :T_BA_StateText:='ULA';
  Recirculating_air_system_sDescription                          :T_BA_StateText:='Umluftanlage';
  Full_air_conditioning_system_sObjectName                      :T_BA_StateText:='VKA';
  Full_air_conditioning_system_sDescription                      :T_BA_StateText:='Vollklimaanlage';
  Heat_recovery_system_sObjectName                              :T_BA_StateText:='WRG';
  Heat_recovery_system_sDescription                              :T_BA_StateText:='Wärmerückgewinnungssystem';
  Intake_air_system_sObjectName                                 :T_BA_StateText:='ZUA';
  Intake_air_system_sDescription                                 :T_BA_StateText:='Zuluftanlage';
  Smoke_extraction_system_sObjectName                           :T_BA_StateText:='ERA';
  Smoke_extraction_system_sDescription                           :T_BA_StateText:='Entrauchungsanlage';
// 434 Kälteanlagen
  Remote_cooling_transfer_sObjectName                           :T_BA_StateText:='FKÜ';
  Remote_cooling_transfer_sDescription                           :T_BA_StateText:='Fernkälteübergabe';
  Cooling_sObjectName                                           :T_BA_StateText:='KAE';
  Cooling_sDescription                                           :T_BA_StateText:='Kälte (allgemein)';
  Cooling_circuit_sObjectName                                   :T_BA_StateText:='KKR';
  Cooling_circuit_sDescription                                   :T_BA_StateText:='Kältekreis';
  Cooling_distribution_network_sObjectName                      :T_BA_StateText:='KVN';
  Cooling_distribution_network_sDescription                      :T_BA_StateText:='Kälteverteilnetz';
  Cold_water_generation_sObjectName                             :T_BA_StateText:='KWE';
  Cold_water_generation_sDescription                             :T_BA_StateText:='Kaltwassererzeugung';
  Electrical_cabinet_cooling_sObjectName                        :T_BA_StateText:='KVE';
  Electrical_cabinet_cooling_sDescription                        :T_BA_StateText:='Kühlung Schaltschrank ';
  Cooling_storage_sObjectName                                   :T_BA_StateText:='KSP';
  Cooling_storage_sDescription                                   :T_BA_StateText:='Kältespeicher';
  Chilled_ceiling_sObjectName                                   :T_BA_StateText:='KÜD';
  Chilled_ceiling_sDescription                                   :T_BA_StateText:='Kühldecke';
  Re_cooling_plant_sObjectName                                  :T_BA_StateText:='RKW';
  Re_cooling_plant_sDescription                                  :T_BA_StateText:='Rückkühlwerk (auch Kühlturm)';
// 441 Hoch- und Mittelspannungsanlagen
  Switchgear_sObjectName                                        :T_BA_StateText:='STA';
  Switchgear_sDescription                                        :T_BA_StateText:='Schaltanlagen';
  Transformer_sObjectName                                       :T_BA_StateText:='TRF';
  Transformer_sDescription                                       :T_BA_StateText:='Transformator';
  Medium_voltage_system_sObjectName                             :T_BA_StateText:='MSA';
  Medium_voltage_system_sDescription                             :T_BA_StateText:='Mittelspannungsanlage';
  Compensation_system_sObjectName                               :T_BA_StateText:='KOA';
  Compensation_system_sDescription                               :T_BA_StateText:='Kompensationsanlage';
  Frequency_converter_system_sObjectName                        :T_BA_StateText:='FUA';
  Frequency_converter_system_sDescription                        :T_BA_StateText:='Frequenzumformeranlage';
// 442 Eigenstromversorgungsanlagen
  Emissions_system_sObjectName                                  :T_BA_StateText:='AGA';
  Emissions_system_sDescription                                  :T_BA_StateText:='Abgasanlage';
  Battery_unit_sObjectName                                      :T_BA_StateText:='BAT';
  Battery_unit_sDescription                                      :T_BA_StateText:='Batterieanlage';
  Co_generation_unit_sObjectName                                :T_BA_StateText:='BHK';
  Co_generation_unit_sDescription                                :T_BA_StateText:='Blockheizkraftwerk';
  Fuel_supply_sObjectName                                       :T_BA_StateText:='BRV';
  Fuel_supply_sDescription                                       :T_BA_StateText:='Brennstoffversorgung';
  Standby_power_system_sObjectName                              :T_BA_StateText:='ESA';
  Standby_power_system_sDescription                              :T_BA_StateText:='Ersatzstromanlage';
  Photovoltaic_system_sObjectName                               :T_BA_StateText:='PVA';
  Photovoltaic_system_sDescription                               :T_BA_StateText:='Fotovoltaikanlage';
  Uninterruptible_power_supply_sObjectName                      :T_BA_StateText:='USV';
  Uninterruptible_power_supply_sDescription                      :T_BA_StateText:='Unterbrechungsfreie Stromversorgung';
// 443 Niederspannungsschaltanlagen
  General_power_supply_sObjectName                              :T_BA_StateText:='ASV';
  General_power_supply_sDescription                              :T_BA_StateText:='Allgemeine Stromversorgung';
  Safety_power_supply_sObjectName                               :T_BA_StateText:='SSV';
  Safety_power_supply_sDescription                               :T_BA_StateText:='Sicherheitsstromversorgung';
  Lighting_sObjectName                                          :T_BA_StateText:='BEL';
  Lighting_sDescription                                          :T_BA_StateText:='Beleuchtungsanlage';
  Emergency_lighting_sObjectName                                :T_BA_StateText:='SIB';
  Emergency_lighting_sDescription                                :T_BA_StateText:='Sicherheitsbeleuchtung';
// 451 Telekommunikationsanlagen
  Telecommunications_system_sObjectName                         :T_BA_StateText:='TEL';
  Telecommunications_system_sDescription                         :T_BA_StateText:='Telekommunikationsanlage';
// 452 Such- und Signalanlagen
  Call_signalling_system_sObjectName                            :T_BA_StateText:='LRA';
  Call_signalling_system_sDescription                            :T_BA_StateText:='Lichtrufanlage';
  Door_intercom_and_door_opener_system_sObjectName              :T_BA_StateText:='TÜA';
  Door_intercom_and_door_opener_system_sDescription              :T_BA_StateText:='Türsprech- und -öffneranlage';
  Paging_system_sObjectName                                     :T_BA_StateText:='PRA';
  Paging_system_sDescription                                     :T_BA_StateText:='Personenrufanlage';
// 453 Zeitdienstanlagen
  Clock_and_time_recording_system_sObjectName                   :T_BA_StateText:='ZEA';
  Clock_and_time_recording_system_sDescription                   :T_BA_StateText:='Uhren- und Zeiterfassungsanlage';
// 454 Elektroakustische Anlagen
  Electro_acoustic_sound_systems_sObjectName                    :T_BA_StateText:='ELA';
  Electro_acoustic_sound_systems_sDescription                    :T_BA_StateText:='Elektroakustische Anl. , Beschallung';
  Conference_and_interpreting_equipment_sObjectName             :T_BA_StateText:='KDA';
  Conference_and_interpreting_equipment_sDescription             :T_BA_StateText:='Konferenz- und Dolmetscheranlage';
  Intercom_system_sObjectName                                   :T_BA_StateText:='GSA';
  Intercom_system_sDescription                                   :T_BA_StateText:='Gegensprechanlage';
  Voice_alarm_system_sObjectName                                :T_BA_StateText:='SAA';
  Voice_alarm_system_sDescription                                :T_BA_StateText:='Sprachalarmierungsanlage';
  Intercommunication_systems_sObjectName                        :T_BA_StateText:='WSA';
  Intercommunication_systems_sDescription                        :T_BA_StateText:='Wechselsprechanlagen';
// 455 Fernseh- und Antennenanlagen
  Television_system_sObjectName                                 :T_BA_StateText:='TVA';
  Television_system_sDescription                                 :T_BA_StateText:='Fernsehanlage';
  Transmitting_and_receiving_antenna_system_sObjectName         :T_BA_StateText:='SEA';
  Transmitting_and_receiving_antenna_system_sDescription         :T_BA_StateText:='Sende- und Empfangsantennenanlage';
  BOS_radio_system_sObjectName                                  :T_BA_StateText:='BOS';
  BOS_radio_system_sDescription                                  :T_BA_StateText:='BOS-Funkanlage';
// 456 Gefahrenmelde- und Alarmanlagen
  Fire_detection_and_alarm_system_sObjectName                   :T_BA_StateText:='BMA';
  Fire_detection_and_alarm_system_sDescription                   :T_BA_StateText:='Brandmeldeanlage';
  Carbon_monoxide_warning_system_sObjectName                    :T_BA_StateText:='COW';
  Carbon_monoxide_warning_system_sDescription                    :T_BA_StateText:='CO-Warnanlage';
  Burglar_alarm_system_sObjectName                              :T_BA_StateText:='EMA';
  Burglar_alarm_system_sDescription                              :T_BA_StateText:='Einbruchmeldeanlage';
  Fire_control_panel_sObjectName                                :T_BA_StateText:='FWT';
  Fire_control_panel_sDescription                                :T_BA_StateText:='Feuerwehrtableau';
  Escape_route_protection_system_sObjectName                    :T_BA_StateText:='FWS';
  Escape_route_protection_system_sDescription                    :T_BA_StateText:='Fluchtwegsicherungsanlage';
  Hazard_detection_system_sObjectName                           :T_BA_StateText:='GMA';
  Hazard_detection_system_sDescription                           :T_BA_StateText:='Gefahrenmeldeanlage';
  Gas_warning_system_sObjectName                                :T_BA_StateText:='GWA';
  Gas_warning_system_sDescription                                :T_BA_StateText:='Gaswarnanlage';
  Smoke_aspiration_system_sObjectName                           :T_BA_StateText:='RAS';
  Smoke_aspiration_system_sDescription                           :T_BA_StateText:='Rauchansaugsystem';
  Room_observation_system_sObjectName                           :T_BA_StateText:='RBA';
  Room_observation_system_sDescription                           :T_BA_StateText:='Raumbeobachtungsanlage';
  Robbery_alarm_system_sObjectName                              :T_BA_StateText:='ÜFA';
  Robbery_alarm_system_sDescription                              :T_BA_StateText:='Überfallmeldeanlage';
  Guard_control_system_sObjectName                              :T_BA_StateText:='WKA';
  Guard_control_system_sDescription                              :T_BA_StateText:='Wächterkontrollanlage';
  Emergency_call_system_sObjectName                             :T_BA_StateText:='NOT';
  Emergency_call_system_sDescription                             :T_BA_StateText:='Notrufanlage';
  Access_control_system_sObjectName                             :T_BA_StateText:='ZKS';
  Access_control_system_sDescription                             :T_BA_StateText:='Zugangskontrollsystem';
// 457 Übertragungsnetze
  Networks_for_the_transmission_voice_text_etc_sObjectName      :T_BA_StateText:='LAN';
  Networks_for_the_transmission_voice_text_etc_sDescription      :T_BA_StateText:='Netzw.  Daten, Sprache, Text etc';
// 459 Fernmelde- und informationstechnische Anlagen, Sonstiges
  Remote_control_systems_sObjectName                            :T_BA_StateText:='FWA';
  Remote_control_systems_sDescription                            :T_BA_StateText:='Fernwirkanlagen';
  Parking_guidance_systems_sObjectName                          :T_BA_StateText:='PLS';
  Parking_guidance_systems_sDescription                          :T_BA_StateText:='Parkleitsysteme';
// 460 Förderanlagen
  File_transportation_systems_sObjectName                       :T_BA_StateText:='ATA';
  File_transportation_systems_sDescription                       :T_BA_StateText:='Aktentransportanlagen';
  Lift_sObjectName                                              :T_BA_StateText:='AUF';
  Lift_sDescription                                              :T_BA_StateText:='Aufzug';
  Inspection_systems_sObjectName                                :T_BA_StateText:='BFA';
  Inspection_systems_sDescription                                :T_BA_StateText:='Befahranlagen';
  Moving_walkways_sObjectName                                   :T_BA_StateText:='FST';
  Moving_walkways_sDescription                                   :T_BA_StateText:='Fahrsteige';
  Escalators_sObjectName                                        :T_BA_StateText:='FTR';
  Escalators_sDescription                                        :T_BA_StateText:='Fahrtreppen';
  External_lifts_sObjectName                                    :T_BA_StateText:='FSA';
  External_lifts_sDescription                                    :T_BA_StateText:='Fassadenaufzüge';
  Baggage_conveyor_system_sObjectName                           :T_BA_StateText:='GFA';
  Baggage_conveyor_system_sDescription                           :T_BA_StateText:='Gepäckförderanlage';
  Pneumatic_delivery_systems_sObjectName                        :T_BA_StateText:='RPA';
  Pneumatic_delivery_systems_sDescription                        :T_BA_StateText:='Rohrpostanlagen';
  Goods_transportation_facilities_sObjectName                   :T_BA_StateText:='WTA';
  Goods_transportation_facilities_sDescription                   :T_BA_StateText:='Warentransportanlagen';
// 470 Nutzerspezifische Anlagen
// 471 Küchentechnische Anlagen
  Small_refrigeration_unit_sObjectName                          :T_BA_StateText:='KLK';
  Small_refrigeration_unit_sDescription                          :T_BA_StateText:='Kleinkälteanlage';
// 472 Wäscherei- und Reinigungsanlagen
  Disinfection_unit_sObjectName                                 :T_BA_StateText:='DES';
  Disinfection_unit_sDescription                                 :T_BA_StateText:='Desinfektionsanlage';
  Cleaning_unit_sObjectName                                     :T_BA_StateText:='REA';
  Cleaning_unit_sDescription                                     :T_BA_StateText:='Reinigungsanlage';
  Sterilisation_systems_sObjectName                             :T_BA_StateText:='STR';
  Sterilisation_systems_sDescription                             :T_BA_StateText:='Sterilisationseinrichtungen';
  Water_treatment_system_sObjectName                            :T_BA_StateText:='WAA';
  Water_treatment_system_sDescription                            :T_BA_StateText:='Wasseraufbereitungsanlage';
  Laundry_system_sObjectName                                    :T_BA_StateText:='WÄA';
  Laundry_system_sDescription                                    :T_BA_StateText:='Wäschereianlage';
// 473 Medienversorgungsanlagen
  Compressed_air_supply_system_sObjectName                      :T_BA_StateText:='DRL';
  Compressed_air_supply_system_sDescription                      :T_BA_StateText:='Druckluftversorgungsanlage';
  Pressure_regulator_unit_sObjectName                           :T_BA_StateText:='DRA';
  Pressure_regulator_unit_sDescription                           :T_BA_StateText:='Druckregelanlage';
  Media_supply_system_sObjectName                               :T_BA_StateText:='MVA';
  Media_supply_system_sDescription                               :T_BA_StateText:='Medienversorgungsanlage';
  Medical_and_technical_gases_sObjectName                       :T_BA_StateText:='MTG';
  Medical_and_technical_gases_sDescription                       :T_BA_StateText:='Medizinische und technische Gase';
  Vacuum_unit_sObjectName                                       :T_BA_StateText:='VAK';
  Vacuum_unit_sDescription                                       :T_BA_StateText:='Vakuumanlage';
// 474 Medizin- und labortechnische Anlagen
  Medical_technical_plant_sObjectName                           :T_BA_StateText:='MED';
  Medical_technical_plant_sDescription                           :T_BA_StateText:='Medizintechnische Anlagen';
  Medical_gas_supply_sObjectName                                :T_BA_StateText:='MGV';
  Medical_gas_supply_sDescription                                :T_BA_StateText:='Medizinische Gasversorgung';
  Laboratory_equipment_sObjectName                              :T_BA_StateText:='LAB';
  Laboratory_equipment_sDescription                              :T_BA_StateText:='Labortechnische Anlagen (allgemein)';
// 475 Feuerlöschanlagen
  Fire_extinguisher_sObjectName                                 :T_BA_StateText:='FLA';
  Fire_extinguisher_sDescription                                 :T_BA_StateText:='Feuerlöschanlage';
  Gas_extinguishing_system_sObjectName                          :T_BA_StateText:='GLA';
  Gas_extinguishing_system_sDescription                          :T_BA_StateText:='Gaslöschanlage';
  Fire_extinguishing_system_sObjectName                         :T_BA_StateText:='LÖS';
  Fire_extinguishing_system_sDescription                         :T_BA_StateText:='Löschanlage (allgemein)';
  Mist_extinguishing_system_sObjectName                         :T_BA_StateText:='NLA';
  Mist_extinguishing_system_sDescription                         :T_BA_StateText:='Nebellöschanlage';
  NOX_system_sObjectName                                        :T_BA_StateText:='NOX';
  NOX_system_sDescription                                        :T_BA_StateText:='NOX-Anlage';
  Sprinkler_system_sObjectName                                  :T_BA_StateText:='SPR';
  Sprinkler_system_sDescription                                  :T_BA_StateText:='Sprinkleranlage';
  Wall_hydrant_system_sObjectName                               :T_BA_StateText:='WHA';
  Wall_hydrant_system_sDescription                               :T_BA_StateText:='Wandhydrantenanlage';
// 478 Entsorgungsanlagen
  Waste_disposal_system_sObjectName                             :T_BA_StateText:='AEA';
  Waste_disposal_system_sDescription                             :T_BA_StateText:='Abfallentsorgungsanlage';
  Media_disposal_system_sObjectName                             :T_BA_StateText:='MEA';
  Media_disposal_system_sDescription                             :T_BA_StateText:='Medienentsorgungsanlage';
  Vacuum_cleaning_systems_sObjectName                           :T_BA_StateText:='SSA';
  Vacuum_cleaning_systems_sDescription                           :T_BA_StateText:='Staubsauganlagen';
// 480 Gebäudeautomation
  Information_focal_point_sObjectName                           :T_BA_StateText:='ISP';
  Information_focal_point_sDescription                           :T_BA_StateText:='Informationsschwerpunkt';
  Weather_station_sObjectName                                   :T_BA_StateText:='WET';
  Weather_station_sDescription                                   :T_BA_StateText:='Wetterstation';
  Management_and_operating_equipment_sObjectName                :T_BA_StateText:='MBE';
  Management_and_operating_equipment_sDescription                :T_BA_StateText:='Management- und Bedieneinrichtungen';
  Room_automation_sObjectName                                   :T_BA_StateText:='RAU';
  Room_automation_sDescription                                   :T_BA_StateText:='Raumautomation';
  Room_automation_system_distributor_sObjectName                :T_BA_StateText:='RAV';
  Room_automation_system_distributor_sDescription                :T_BA_StateText:='Raumautomation-Systemverteiler';
  Control_cabinet_sObjectName                                   :T_BA_StateText:='SSK';
  Control_cabinet_sDescription                                   :T_BA_StateText:='Schaltschrank';
  Settings_sObjectName                                          :T_BA_StateText:='ALP';
  Settings_sDescription                                          :T_BA_StateText:='Anlagenparameter';
  EventGroups_sObjectName                                       :T_BA_StateText:='ERG';
  EventGroups_sDescription                                       :T_BA_StateText:='Meldeklassen';
  Global_Building_Data_sObjectName                              :T_BA_StateText:='GGL';
  Global_Building_Data_sDescription                              :T_BA_StateText:='globale Gebäudedaten';
// 540 Technische Anlagen in Außenanlagen
  Rainwater_retention_basin_sObjectName                         :T_BA_StateText:='RRB';
  Rainwater_retention_basin_sDescription                         :T_BA_StateText:='Regenrückhaltebecken';
  Cistern_system_sObjectName                                    :T_BA_StateText:='ZTA';
  Cistern_system_sDescription                                    :T_BA_StateText:='Zisternenanlage';
END_VAR

// ---- Templates/GVLs/DPAD/Texts/TextTrades.TcGVL
{region '#Template'}
	{attribute 'Version' := '0.0.1.0'}
	{attribute 'Tags' := '"LCID": "1031", "Text": "GVL, DPAD, Trades, ObjectName, Description"'}
	{attribute 'Tags' := '"LCID": "1033", "Text": "GVL, DPAD, Trades, ObjectName, Description"'}
	{attribute 'Description' := '"LCID": "1031", "Text": "Textliste Gewerke"'}
	{attribute 'Description' := '"LCID": "1033", "Text": "Text list trades"'}
{endregion}

{attribute 'qualified_only'}
{attribute 'global_init_slot' := '40510'}
// generated:21.05.2021 -- 09:43:24 list with plant descriptions
VAR_GLOBAL
  Doors_gates_windows_sun_protection_sObjectName                :T_BA_StateText:='Doors, gates, windows, sun protection';
  Doors_gates_windows_sun_protection_sDescription                :T_BA_StateText:='DGW';
  Sewage_water_and_gas_plants_sObjectName                       :T_BA_StateText:='Sewage, water and gas plants';
  Sewage_water_and_gas_plants_sDescription                       :T_BA_StateText:='SWG';
  Heat_supply_systems_sObjectName                               :T_BA_StateText:='Heat supply systems';
  Heat_supply_systems_sDescription                               :T_BA_StateText:='HTG';
  Air_conditioning_sObjectName                                  :T_BA_StateText:='Air conditioning';
  Air_conditioning_sDescription                                  :T_BA_StateText:='AC_';
  Refrigeration_systems_sObjectName                             :T_BA_StateText:='Refrigeration systems';
  Refrigeration_systems_sDescription                             :T_BA_StateText:='RFG';
  High_voltage_systems_sObjectName                              :T_BA_StateText:='High-voltage systems';
  High_voltage_systems_sDescription                              :T_BA_StateText:='HVS';
  Telecommunication_and_information_technology_sObjectName      :T_BA_StateText:='Telecom. and information tech. equipment';
  Telecommunication_and_information_technology_sDescription      :T_BA_StateText:='TIT';
  Hazard_detection_and_alarm_systems_sObjectName                :T_BA_StateText:='Hazard detection and alarm systems';
  Hazard_detection_and_alarm_systems_sDescription                :T_BA_StateText:='HDA';
  Conveyors_sObjectName                                         :T_BA_StateText:='Conveyors';
  Conveyors_sDescription                                         :T_BA_StateText:='CVY';
  Kitchen_technology_systems_sObjectName                        :T_BA_StateText:='Kitchen technology systems';
  Kitchen_technology_systems_sDescription                        :T_BA_StateText:='KTS';
  Laundry_and_cleaning_systems_sObjectName                      :T_BA_StateText:='Laundry and cleaning systems';
  Laundry_and_cleaning_systems_sDescription                      :T_BA_StateText:='LCS';
  Media_supply_systems_sObjectName                              :T_BA_StateText:='Media supply systems';
  Media_supply_systems_sDescription                              :T_BA_StateText:='MSS';
  Medical_and_laboratory_equipment_sObjectName                  :T_BA_StateText:='Medical and laboratory equipment';
  Medical_and_laboratory_equipment_sDescription                  :T_BA_StateText:='MED';
  Fire_extinguishing_systems_sObjectName                        :T_BA_StateText:='Fire extinguishing systems';
  Fire_extinguishing_systems_sDescription                        :T_BA_StateText:='FES';
  Bathing_facilities_sObjectName                                :T_BA_StateText:='Bathing facilities';
  Bathing_facilities_sDescription                                :T_BA_StateText:='BTF';
  Process_heating_cooling_and_air_systems_sObjectName           :T_BA_StateText:='Process heating, cooling and air systems';
  Process_heating_cooling_and_air_systems_sDescription           :T_BA_StateText:='PRO';
  Waste_disposal_facilities_sObjectName                         :T_BA_StateText:='Waste disposal facilities';
  Waste_disposal_facilities_sDescription                         :T_BA_StateText:='WDF';
  Building_automation_and_control_systems_general_sObjectName   :T_BA_StateText:='Building automation  general';
  Building_automation_and_control_systems_general_sDescription   :T_BA_StateText:='BAG';
  Automation_focal_point_information_focal_point_sObjectName    :T_BA_StateText:='Automation focal point';
  Automation_focal_point_information_focal_point_sDescription    :T_BA_StateText:='AFP';
  Room_automation_sObjectName                                   :T_BA_StateText:='Room automation';
  Room_automation_sDescription                                   :T_BA_StateText:='ROM';
  Outdoor_devices_sObjectName                                   :T_BA_StateText:='Outdoor devices';
  Outdoor_devices_sDescription                                   :T_BA_StateText:='ODD';
END_VAR

// ---- POUs/MAIN.TcPOU
PROGRAM MAIN
VAR
	DPAD		: FB_BA_CarelessDPAD := (
					aIdentifier := [
	(* Level 1 *)		(eMode:=E_BA_DPADMode.eInclude,		eNodeType:=E_BA_NodeType.eLocation,			sSeparator_ObjectName := '_', 	sSeparator_Description := ' - ',	nIndexDigits := 0),
	(* Level 2 *)		(eMode:=E_BA_DPADMode.eInclude,		eNodeType:=E_BA_NodeType.eBuilding,			sSeparator_ObjectName := '_', 	sSeparator_Description := ' - ',	nIndexDigits := 0),
	(* Level 3 *)		(eMode:=E_BA_DPADMode.eInclude,		eNodeType:=E_BA_NodeType.eControlCabinet,	sSeparator_ObjectName := '_', 	sSeparator_Description := ' - ',	nIndexDigits := 0),
	(* Level 4 *)		(eMode:=E_BA_DPADMode.eInclude,		eNodeType:=E_BA_NodeType.eFloor,			sSeparator_ObjectName := '_', 	sSeparator_Description := ' - ',	nIndexDigits := 0),
	(* Level 5 *)		(eMode:=E_BA_DPADMode.eInclude,		eNodeType:=E_BA_NodeType.eTrade,			sSeparator_ObjectName := '_', 	sSeparator_Description := ' - ',	nIndexDigits := 0),
	(* Level 6 *)		(eMode:=E_BA_DPADMode.eInclude,		eNodeType:=E_BA_NodeType.ePlant,			sSeparator_ObjectName := '=', 	sSeparator_Description := ' = ',	nIndexDigits := 2),
	(* Level 7 *)		(eMode:=E_BA_DPADMode.eInclude,		eNodeType:=E_BA_NodeType.eAggregate,		sSeparator_ObjectName := '-', 	sSeparator_Description := ' - ',	nIndexDigits := 2),
	(* Level 8 *)		(eMode:=E_BA_DPADMode.eInclude,		eNodeType:=E_BA_NodeType.eFunction,			sSeparator_ObjectName := '-', 	sSeparator_Description := ' - ',	nIndexDigits := 2)
					]
				);		
		 
//	Level 1 Standort bzw. Ort oder Stadt 
//	Level 1 Site respectively location or town
	SiteA						: FB_BA_View	:= (sDescription:='Location'	)		;	
//	Level 2 Gebäude 	
//	Level 2 Building 	
		B						: FB_BA_View := 	(iParent := SiteA,	sDescription:='Building'	);     
// Level 3 ISP -> Informationsschwerpunkt
// Level 3 information focal point 	 	                                                                                   	
			IFP01				: FB_BA_View := 	(iParent := B, 		sDescription:='PLC'	);     
// Level 4 Stockwerk 	->	O01 = Obergeschoss 01, U01 = Untergeschoss 01,  E00 = Ergeschoss
// Level 4 floor ->	F01 = floor 01, B01 = basement 01,  GFL = Ground floor  						
				F01				: FB_BA_View := 	(iParent := IFP01, 	sDescription:='Floor 01'	);     	
// Level 5 Gewerk Wärmeversorgungsanlagen  
// Level 5 Trade Heat supply systems, heat distribution  --> 	HD = heat distribution, HG = heat generation
					H			: FB_BA_H 	:= 		(iParent := F01, 	sDescription:='Heating'	);     	 															   	 	
// Level 5 Gewerk Gebäudeautomation Allgemein   
// Level 5 Trade General                                                                                       	
					G			: FB_BA_General := 	(iParent := F01, 	sDescription:='General'	);     	 											
// Level 5 Gewerk Luftechnische Anlagen      
// Level 5 Trade ventilation system                                                                                	
					AC			: FB_BA_AC 		:= 	(iParent := F01, 	sDescription:='AirCondition'	);     	   	
// Level 5 Gewerk Raumautomation    
// Level 5 Trade room automation                                                                              	
				
//	Test Level
					WeatherStation	: FB_BA_WeatherStation := (iParent			:= F01, sDescription:='Weatherstation'	); 					
END_VAR

//	Level 1 Standort bzw. Ort oder Stadt 
SiteA();

//	Level 2 Gebäude 		
	B();

// Level 3 ISP -> Informationsschwerpunkt
		IFP01();

// Level 4 Stockwerk -->	O01 = Obergeschoss 01, U01 = Untergeschoss 01,  E00 = Ergeschoss 
			F01();

// Level 5 Gewerk Wärmeversorgungsanlagen	
				H();								
// Level 5 Gewerk Allgemein				
				G(); 								
// Level 5 Gewerk Luftechnische Anlagen		
				AC();								
// Level 5 Gewerk Raumautomation 
					
// Level 5 Test
				WeatherStation();

METHOD FB_init : BOOL
VAR_INPUT
	bInitRetains : BOOL; // if TRUE, the retain variables are initialized (warm start / cold start)
	bInCopyCode : BOOL;  // if TRUE, the instance afterwards gets moved into the copy code (online change)
END_VAR
END_METHOD

END_PROGRAM

// ---- Templates/POUs/Trade/AC/Aggregates/Cooler/Temperature/FB_BA_AC_ColTSuACtrl.TcPOU
{region '#Template'}
	{attribute 'Version' := '1.0.0.0'}
	{attribute 'Tags' := '"LCID": "1031", "Text": "AC, Aggregates, Cooler, Temperature, Controller"'}
	{attribute 'Tags' := '"LCID": "1033", "Text": "AC, Aggregates, Cooler, Temperature, Controller"'}
	{attribute 'Description' := '"LCID": "1031", "Text": "Kühler Zuluft Regler Temperatur"'}
	{attribute 'Description' := '"LCID": "1033", "Text": "Cooler Supply air controller temperature"'}
{endregion}
FUNCTION_BLOCK FB_BA_AC_ColTSuACtrl EXTENDS FB_BA_View
VAR_INPUT
	bEn						: BOOL;
	fSpTSuA					: REAL;// Sollwert Temperatur kühlen // Setpoint temperature cooling
	fTSuA					: REAL;// Zuluft Temperatur // Supply air temperature
	bSync					: BOOL;
	fSync					: REAL;
END_VAR
VAR_OUTPUT
	fY              		: REAL;
	bIsActive				: BOOL;	//	active sequence controller
	bOpState				: BOOL;	//	Release sequence link, sequence control is active	
END_VAR
VAR_INPUT CONSTANT
	Ctrl					: FB_BA_Loop;
END_VAR

SUPER^(); // FB_BA_View
Ctrl(bEn := bEn, fSetpoint := fSpTSuA, fCtrlVal := fTSuA, bEnSync := bSync, fValSync := fSync); // FB_BA_Loop
fY := Ctrl.fPresentValue;
bOpState := Ctrl.OpState;
bIsActive := Ctrl.IsActive;

METHOD FB_init : BOOL
VAR_INPUT
	bInitRetains : BOOL; // if TRUE, the retain variables are initialized (warm start / cold start)
	bInCopyCode : BOOL;  // if TRUE, the instance afterwards gets moved into the copy code (online change)
END_VAR
Ctrl.iParent						:= THIS^;
Ctrl.iLabel							:= LblCmpAC.Cooler_TSuACtrl_Ctrl; 
Ctrl.sObjectName					:= '{Idx=01}';
Ctrl.eOpMode						:= BA2_Param.nLoop_DefOpMode;								 	 										 
Ctrl.eOutputUnit					:= E_BA_Unit.eOther_Percent;
Ctrl.eActionRm						:= E_BA_Action.eDirect;
Ctrl.fProportionalConstant			:= 3;
Ctrl.fIntegralConstant				:= 180;
Ctrl.fDerivativeConstant			:= 0;
Ctrl.fMaxOutputRm 					:= 100;
Ctrl.fMinOutputRm					:= 0;
Ctrl.fCOVIncrement					:= 0;
Ctrl.nDampConstant					:= 0;
Ctrl.fNeutralZone					:= 0;
END_METHOD

END_FUNCTION_BLOCK

// ---- Templates/POUs/Trade/AC/General/FB_BA_AC_OpMod1St.TcPOU
{region '#Template'}
	{attribute 'Version' := '1.0.0.0'}
	{attribute 'Tags' := '"LCID": "1031", "Text": "AC, General, AHU, Operating mode"'}
	{attribute 'Tags' := '"LCID": "1033", "Text": "AC, General, AHU, Operating mode"'}
	{attribute 'Description' := '"LCID": "1031", "Text": "Betriebsart"'}
	{attribute 'Description' := '"LCID": "1033", "Text": "Operating mode"'}
{endregion}
FUNCTION_BLOCK FB_BA_AC_OpMod1St EXTENDS FB_BA_View
VAR_INPUT
	bSmExttSuA				: BOOL;	// smoke extraction supply air
	bSmExttExhA				: BOOL;	// smoke extraction exhaust air
	bFireDetc				: BOOL;	// fire detection alarm
	bForcVent				: BOOL;	// Forced ventilation
	bEmgOff					: BOOL;	// emergency stop
	bFrst					: BOOL;	// Frost protection is active
	bCentSwiOff				: BOOL;	// Central switch-off	
	bAlmShutOff				: BOOL;	// Shut Off plant collective alarm
	bNgtCol					: BOOL;	// Summer night cooling
	bColDwnPrtc				: BOOL;	// Cooling down protection
	bOvrHtgPrtc				: BOOL;	// Overheating protection
END_VAR
VAR_OUTPUT
	eOpMode					: E_BA_AC_OpMod01;
END_VAR
VAR_INPUT CONSTANT
	OpModMan				: FB_BA_MV_Op;	
	Sched					: FB_BA_SchedM;
	OpModPr					: FB_BA_MV_Op;
END_VAR
VAR
	PrioSwi					: FB_BA_PrioSwi_UDI24;
END_VAR

SUPER^(); // FB_BA_View
OpModMan(); // FB_BA_MV_Op
Sched(); // FB_BA_SchedM
PrioSwi(
    bEn02 := bSmExttSuA AND bSmExttExhA,
    nVal02 := E_BA_AC_OpMod01.eSmokeExtractionProgramm,
    bEn03 := bSmExttSuA,
    nVal03 := E_BA_AC_OpMod01.eSmokeExtractionSupplyAir,
    bEn04 := bSmExttExhA,
    nVal04 := E_BA_AC_OpMod01.eSmokeExtractionExhaustAir,
    bEn05 := bFireDetc,
    nVal05 := E_BA_AC_OpMod01.eFire,
    bEn07 := bForcVent,
    nVal07 := E_BA_AC_OpMod01.eForcedVentilation,
    bEn08 := bEmgOff,
    nVal08 := E_BA_AC_OpMod01.eEmergency,
    bEn09 := bFrst,
    nVal09 := E_BA_AC_OpMod01.eFrost,
    bEn10 := bCentSwiOff,
    nVal10 := E_BA_AC_OpMod01.eCentralSwitchOff,
    bEn11 := bAlmShutOff,
    nVal11 := E_BA_AC_OpMod01.eAlarm,
    bEn14 := E_BA_OnOffA.eOff = OpModMan.nPresentValue,
    nVal14 := E_BA_AC_OpMod01.eOff,
    bEn15 := OpModMan.nPresentValue = E_BA_OnOffA.eOn,
    nVal15 := E_BA_AC_OpMod01.eOn,
    bEn18 := Sched.nPresentValue = E_BA_OnOff.eOn,
    nVal18 := E_BA_AC_OpMod01.eOn,
    bEn20 := bNgtCol,
    nVal20 := E_BA_AC_OpMod01.eNightCooling,
    bEn21 := bColDwnPrtc,
    nVal21 := E_BA_AC_OpMod01.eCoolDownProtection,
    bEn22 := bOvrHtgPrtc,
    nVal22 := E_BA_AC_OpMod01.eOverHeatingProtection,
    bEn24 := TRUE,
    nVal24 := E_BA_AC_OpMod01.eOFF); // FB_BA_PrioSwi_UDI24
OpModPr(nValuePgm := PrioSwi.nVal); // FB_BA_MV_Op
eOpMode := OpModPr.nPresentValue;

METHOD FB_init : BOOL
VAR_INPUT
	bInitRetains : BOOL; // if TRUE, the retain variables are initialized (warm start / cold start)
	bInCopyCode : BOOL;  // if TRUE, the instance afterwards gets moved into the copy code (online change)
END_VAR
OpModMan.iParent			:= THIS^;
OpModMan.iLabel				:= LblCmpAC.General_OpModMan;							
OpModMan.sObjectName		:= '{Idx=01}';								 	 
OpModMan.aStateText[1]		:= txtEvent_Auto;
OpModMan.aStateText[2]		:= txtEvent_Off;
OpModMan.aStateText[3]		:= txtEvent_On;
OpModMan.nValueRm			:= E_BA_OnOffA.eAutomatic;

OpModPr.iParent				:= THIS^;
OpModPr.iLabel				:= LblCmpAC.General_OpModPr;							
OpModPr.sObjectName			:= '{Idx=01}';								 	 
OpModPr.aStateText[1]		:= txtEvent_Off;
OpModPr.aStateText[2]		:= txtEvent_On;
OpModPr.aStateText[3]		:= txtEvent_EmergencyStop;
OpModPr.aStateText[4]		:= txtEvent_Frost;
OpModPr.aStateText[5]		:= txtEvent_SmokeExtraction_P;
OpModPr.aStateText[6]		:= txtEvent_SmokeExtractionSupplyAir;
OpModPr.aStateText[7]		:= txtEvent_SmokeExtractionExtractAir;
OpModPr.aStateText[8]		:= txtEvent_Fire;
OpModPr.aStateText[9]		:= txtEvent_NightCooling;
OpModPr.aStateText[10]		:= txtEvent_CoolDownProtection;
OpModPr.aStateText[11]		:= txtEvent_OverHeatingProtection;
OpModPr.aStateText[12]		:= txtEvent_Disturb;
OpModPr.aStateText[13]		:= txtEvent_ForcedVentilation;
OpModPr.aStateText[14]		:= txtEvent_CentralSwitchOff; 		

Sched.iParent											:= THIS^;
Sched.iLabel											:= LblCmpAC.General_Sched;							
Sched.sObjectName										:= '{Idx=01}';		
Sched.aStateText[1]										:= txtEvent_Off;
Sched.aStateText[2]										:= txtEvent_On;
Sched.nPredictTime										:= 0;
Sched.nDefaultValue										:= E_BA_OnOff.eOff;
Sched.bWriteWeekly										:= FALSE;
//	Monday
Sched.aWeek[E_BA_Weekday.eMonday,1].eState				:= E_BA_SchedEntryState.eValue;
Sched.aWeek[E_BA_Weekday.eMonday,1].uValue.udiVal		:= E_BA_OnOff.eOn;
Sched.aWeek[E_BA_Weekday.eMonday,1].stTime.nHour		:= 6;
Sched.aWeek[E_BA_Weekday.eMonday,1].stTime.nMinute		:= 0;
Sched.aWeek[E_BA_Weekday.eMonday,1].stTime.nSecond		:= 0;
Sched.aWeek[E_BA_Weekday.eMonday,2].eState				:= E_BA_SchedEntryState.eValue;
Sched.aWeek[E_BA_Weekday.eMonday,2].uValue.udiVal		:= E_BA_OnOff.eOff;
Sched.aWeek[E_BA_Weekday.eMonday,2].stTime.nHour		:= 20;
Sched.aWeek[E_BA_Weekday.eMonday,2].stTime.nMinute		:= 0;
Sched.aWeek[E_BA_Weekday.eMonday,2].stTime.nSecond		:= 0;
Sched.aWeek[E_BA_Weekday.eMonday,3].eState				:= E_BA_SchedEntryState.eValue;
Sched.aWeek[E_BA_Weekday.eMonday,3].uValue.udiVal		:= E_BA_OnOff.eOff;
Sched.aWeek[E_BA_Weekday.eMonday,3].stTime.nHour		:= 0;
Sched.aWeek[E_BA_Weekday.eMonday,3].stTime.nMinute		:= 0;
Sched.aWeek[E_BA_Weekday.eMonday,3].stTime.nSecond		:= 0;
//	Tuesday
Sched.aWeek[E_BA_Weekday.eTuesday,1].eState				:= E_BA_SchedEntryState.eValue;
Sched.aWeek[E_BA_Weekday.eTuesday,1].uValue.udiVal		:= E_BA_OnOff.eOn;
Sched.aWeek[E_BA_Weekday.eTuesday,1].stTime.nHour		:= 6;
Sched.aWeek[E_BA_Weekday.eTuesday,1].stTime.nMinute		:= 0;
Sched.aWeek[E_BA_Weekday.eTuesday,1].stTime.nSecond		:= 0;
Sched.aWeek[E_BA_Weekday.eTuesday,2].eState				:= E_BA_SchedEntryState.eValue;
Sched.aWeek[E_BA_Weekday.eTuesday,2].uValue.udiVal		:= E_BA_OnOff.eOff;
Sched.aWeek[E_BA_Weekday.eTuesday,2].stTime.nHour		:= 20;
Sched.aWeek[E_BA_Weekday.eTuesday,2].stTime.nMinute		:= 0;
Sched.aWeek[E_BA_Weekday.eTuesday,2].stTime.nSecond		:= 0;
Sched.aWeek[E_BA_Weekday.eTuesday,3].eState				:= E_BA_SchedEntryState.eValue;
Sched.aWeek[E_BA_Weekday.eTuesday,3].uValue.udiVal		:= E_BA_OnOff.eOff;
Sched.aWeek[E_BA_Weekday.eTuesday,3].stTime.nHour		:= 0;
Sched.aWeek[E_BA_Weekday.eTuesday,3].stTime.nMinute		:= 0;
Sched.aWeek[E_BA_Weekday.eTuesday,3].stTime.nSecond		:= 0;
//	Wednesday
Sched.aWeek[E_BA_Weekday.eWednesday,1].eState			:= E_BA_SchedEntryState.eValue;
Sched.aWeek[E_BA_Weekday.eWednesday,1].uValue.udiVal	:= E_BA_OnOff.eOn;
Sched.aWeek[E_BA_Weekday.eWednesday,1].stTime.nHour		:= 6;
Sched.aWeek[E_BA_Weekday.eWednesday,1].stTime.nMinute	:= 0;
Sched.aWeek[E_BA_Weekday.eWednesday,1].stTime.nSecond	:= 0;
Sched.aWeek[E_BA_Weekday.eWednesday,2].eState			:= E_BA_SchedEntryState.eValue;
Sched.aWeek[E_BA_Weekday.eWednesday,2].uValue.udiVal	:= E_BA_OnOff.eOff;
Sched.aWeek[E_BA_Weekday.eWednesday,2].stTime.nHour		:= 20;
Sched.aWeek[E_BA_Weekday.eWednesday,2].stTime.nMinute	:= 0;
Sched.aWeek[E_BA_Weekday.eWednesday,2].stTime.nSecond	:= 0;
Sched.aWeek[E_BA_Weekday.eWednesday,3].eState			:= E_BA_SchedEntryState.eValue;
Sched.aWeek[E_BA_Weekday.eWednesday,3].uValue.udiVal	:= E_BA_OnOff.eOff;
Sched.aWeek[E_BA_Weekday.eWednesday,3].stTime.nHour		:= 0;
Sched.aWeek[E_BA_Weekday.eWednesday,3].stTime.nMinute	:= 0;
Sched.aWeek[E_BA_Weekday.eWednesday,3].stTime.nSecond	:= 0;
//	Thursday
Sched.aWeek[E_BA_Weekday.eThursday,1].eState			:= E_BA_SchedEntryState.eValue;
Sched.aWeek[E_BA_Weekday.eThursday,1].uValue.udiVal		:= E_BA_OnOff.eOn;
Sched.aWeek[E_BA_Weekday.eThursday,1].stTime.nHour		:= 6;
Sched.aWeek[E_BA_Weekday.eThursday,1].stTime.nMinute	:= 0;
Sched.aWeek[E_BA_Weekday.eThursday,1].stTime.nSecond	:= 0;
Sched.aWeek[E_BA_Weekday.eThursday,2].eState			:= E_BA_SchedEntryState.eValue;
Sched.aWeek[E_BA_Weekday.eThursday,2].uValue.udiVal		:= E_BA_OnOff.eOff;
Sched.aWeek[E_BA_Weekday.eThursday,2].stTime.nHour		:= 20;
Sched.aWeek[E_BA_Weekday.eThursday,2].stTime.nMinute	:= 0;
Sched.aWeek[E_BA_Weekday.eThursday,2].stTime.nSecond	:= 0;
Sched.aWeek[E_BA_Weekday.eThursday,3].eState			:= E_BA_SchedEntryState.eValue;
Sched.aWeek[E_BA_Weekday.eThursday,3].uValue.udiVal		:= E_BA_OnOff.eOff;
Sched.aWeek[E_BA_Weekday.eThursday,3].stTime.nHour		:= 0;
Sched.aWeek[E_BA_Weekday.eThursday,3].stTime.nMinute	:= 0;
Sched.aWeek[E_BA_Weekday.eThursday,3].stTime.nSecond	:= 0;
//	Friday
Sched.aWeek[E_BA_Weekday.eFriday,1].eState				:= E_BA_SchedEntryState.eValue;
Sched.aWeek[E_BA_Weekday.eFriday,1].uValue.udiVal		:= E_BA_OnOff.eOn;
Sched.aWeek[E_BA_Weekday.eFriday,1].stTime.nHour		:= 6;
Sched.aWeek[E_BA_Weekday.eFriday,1].stTime.nMinute		:= 0;
Sched.aWeek[E_BA_Weekday.eFriday,1].stTime.nSecond		:= 0;
Sched.aWeek[E_BA_Weekday.eFriday,2].eState				:= E_BA_SchedEntryState.eValue;
Sched.aWeek[E_BA_Weekday.eFriday,2].uValue.udiVal		:= E_BA_OnOff.eOff;
Sched.aWeek[E_BA_Weekday.eFriday,2].stTime.nHour		:= 20;
Sched.aWeek[E_BA_Weekday.eFriday,2].stTime.nMinute		:= 0;
Sched.aWeek[E_BA_Weekday.eFriday,2].stTime.nSecond		:= 0;
Sched.aWeek[E_BA_Weekday.eFriday,3].eState				:= E_BA_SchedEntryState.eValue;
Sched.aWeek[E_BA_Weekday.eFriday,3].uValue.udiVal		:= E_BA_OnOff.eOff;
Sched.aWeek[E_BA_Weekday.eFriday,3].stTime.nHour		:= 0;
Sched.aWeek[E_BA_Weekday.eFriday,3].stTime.nMinute		:= 0;
Sched.aWeek[E_BA_Weekday.eFriday,3].stTime.nSecond		:= 0;
Sched.bWriteException									:= FALSE;
END_METHOD

END_FUNCTION_BLOCK

// ---- Templates/POUs/Trade/General/IFP/Project/FB_BA_ProjectEx.TcPOU
{region '#Template'}
	{attribute 'Version' := '0.0.1.0'}
	{attribute 'Tags' := '"LCID": "1031", "Text": "General, Settings, Project, Basics"'}
	{attribute 'Tags' := '"LCID": "1033", "Text": "General, Settings, Project, Basics"'}
	{attribute 'Description' := '"LCID": "1031", "Text": "Projektspezifische Informationen"'}
	{attribute 'Description' := '"LCID": "1033", "Text": "Project specific informations"'}
{endregion}
FUNCTION_BLOCK FB_BA_ProjectEx EXTENDS FB_BA_Project
VAR_INPUT CONSTANT PERSISTENT
	{attribute 'parameterCategory' := 'Persistent Data'}
	tPrsData_DefaultPeriod : TIME := T#30M;
	{attribute 'parameterCategory' := 'Persistent Data'}
	tPrsData_ComissioningPeriod : TIME := T#5M;
	
	{attribute 'parameterCategory' := 'UPS'}
	eUPS : E_BA_UPSType := E_BA_UPSType.eNone;			  
END_VAR
VAR_INPUT CONSTANT
	{attribute 'parameterCategory' := 'Persistent Data'}
	bPrsData_ManualWriteData : BOOL;
END_VAR
VAR_OUTPUT
	nPrsDataWritten			: UINT;
	bPowerFail				: BOOL;
END_VAR
VAR
	_bTriggerUPS			: BOOL;
END_VAR

SUPER^();

UPS();
PersistentData();

METHOD PROTECTED OnInitCycle
VAR
	_stVersion		: ST_LibVersion;
END_VAR
VAR CONSTANT
	FORMAT			: STRING		:= '%d.%d.%d.%d';
END_VAR
CASE (State) OF
	E_BA_ObjectState.eInstanceInit1:
		// Refresh runtime information:
		//_stVersion := F_GetVersion();
		//_stVersion := stLibVersion_BA2_Templates;
		
		BA_Globals.Format(
			pFormatString := ADR(FORMAT),
			arg1:=F_UINT(_stVersion.iMajor),
			arg2:=F_UINT(_stVersion.iMinor),
			arg3:=F_UINT(_stVersion.iBuild),
			arg4:=F_UINT(_stVersion.iRevision),
		
			pDstString := ADR(stVersion.Project),
			nDstSize := SIZEOF(stVersion.Project)
		);
END_CASE

SUPER^();
END_METHOD

METHOD PROTECTED PersistentData
VAR_INST
	nOnlineChangeCnt		:	UDINT;
	iStep					:	INT;
	fbTon					:	TON;
	fbResetOnlineChange		:	TON;
	rtigManual				:	R_TRIG;
	trigUPS					:	R_TRIG;
	rFinishTrig				:	R_TRIG;
	WrtPersistDat			:	FB_BA_WrtPersistDat;
END_VAR
VAR CONSTANT
	DETECT_COMISSIONING_DURATION : TIME := T#60M;
END_VAR
IF	TwinCAT_SystemInfoVarList._AppInfo.OnlineChangeCnt <> nOnlineChangeCnt THEN
	nOnlineChangeCnt := TwinCAT_SystemInfoVarList._AppInfo.OnlineChangeCnt;
	fbResetOnlineChange(IN := FALSE);
	fbTon(IN := FALSE);
	iStep := 10;
END_IF

IF	tPrsData_DefaultPeriod < T#600S THEN
	tPrsData_DefaultPeriod	:= T#1800S;
END_IF

IF	tPrsData_ComissioningPeriod < T#30S THEN
	tPrsData_ComissioningPeriod	:= T#300S;
END_IF

CASE	iStep	OF
	0:
		fbTon(IN := NOT fbTon.Q,PT := tPrsData_DefaultPeriod);
	10:
		fbTon(IN := NOT fbTon.Q,PT := tPrsData_ComissioningPeriod);
		fbResetOnlineChange(IN := TRUE, PT := DETECT_COMISSIONING_DURATION);
		
		IF	fbResetOnlineChange.Q THEN
			iStep := 0;
			fbResetOnlineChange(IN := FALSE);
		END_IF
END_CASE
 
rtigManual(CLK := bPrsData_ManualWriteData);
bPrsData_ManualWriteData := FALSE;

trigUPS(CLK := _bTriggerUPS);

// Write persistent data:
WrtPersistDat(bStt:=(fbTon.Q OR rtigManual.Q OR trigUPS.Q));
rFinishTrig(CLK:=(WrtPersistDat.bBusy AND NOT WrtPersistDat.bErr));

IF (rFinishTrig.Q) THEN
	nPrsDataWritten := (nPrsDataWritten+1);
END_IF
END_METHOD

METHOD PROTECTED UPS
VAR_INST
	fbCX50x0			:	FB_S_UPS;
	fbCX51x0			:	FB_S_UPS_CX51x0;
	fbCX81xx			:	FB_S_UPS_CX81xx;
	fbCX9020_U900		:	FB_S_UPS_CX9020_U900;
	fbCB3011			:	FB_S_UPS_CB3011;
END_VAR
CASE eUPS OF
	E_BA_UPSType.eNone:
		;

	E_BA_UPSType.eCX50x0:
		fbCX50x0(
			sNetID:= '', 
		//	iPLCPort:= TwinCAT_SystemInfoVarList._AppInfo.AdsPort, 
			iUPSPort:= 16#4A8, 
			tTimeout:= DEFAULT_ADS_TIMEOUT, 
			eUpsMode:= eSUPS_CheckPowerStatus, 
			ePersistentMode:= SPDM_2PASS, 
			tRecoverTime:= T#10S, 
			bPowerFailDetect=> bPowerFail, 
			eState=> );

	E_BA_UPSType.eCX51x0:
		fbCX51x0(
			sNetID:= '', 
			iPLCPort:= TwinCAT_SystemInfoVarList._AppInfo.AdsPort, 
			iUPSPort:= 16#588, 
			tTimeout:= DEFAULT_ADS_TIMEOUT, 
			eUpsMode:= eSUPS_CheckPowerStatus, 
			ePersistentMode:= SPDM_2PASS, 
			tRecoverTime:= T#10S, 
			bPowerFailDetect=> bPowerFail, 
			eState=> );

	E_BA_UPSType.eCX81xx:
		fbCX81xx(
			sNetID:= '', 
			iPLCPort:= TwinCAT_SystemInfoVarList._AppInfo.AdsPort, 
			tTimeout:= DEFAULT_ADS_TIMEOUT, 
			eUpsMode:= eSUPS_CheckPowerStatus, 
			ePersistentMode:= SPDM_2PASS, 
			tRecoverTime:= T#10S, 
			bPowerFailDetect=> bPowerFail, 
			eState=> );
		
	E_BA_UPSType.eCX9020_U900:
		fbCX9020_U900(
			sNetID:= '', 
			iPLCPort:= TwinCAT_SystemInfoVarList._AppInfo.AdsPort, 
			tTimeout:= DEFAULT_ADS_TIMEOUT, 
			eUpsMode:= eSUPS_CheckPowerStatus, 
			ePersistentMode:= SPDM_2PASS, 
			tRecoverTime:= T#10S, 
			bPowerFailDetect=> bPowerFail, 
			eState=> );

	E_BA_UPSType.eCB3011:
		fbCB3011(
			sNetID:= '', 
			iPLCPort:= TwinCAT_SystemInfoVarList._AppInfo.AdsPort, 
			tTimeout:= DEFAULT_ADS_TIMEOUT, 
			eUpsMode:= eSUPS_CheckPowerStatus, 
			ePersistentMode:= SPDM_2PASS, 
			tRecoverTime:= T#10S, 
			bPowerFailDetect=> bPowerFail, 
			eState=> );
ELSE
	eUPS := E_BA_UPSType.eNone; 	
END_CASE
END_METHOD

END_FUNCTION_BLOCK

// ---- Templates/POUs/Trade/HeatingSystem/General/FB_BA_H_OpMod.TcPOU
{region '#Template'}
	{attribute 'Version' := '1.0.0.0'}
	{attribute 'Tags' := '"LCID": "1031", "Text": "H, General, HtgCir, Operating mode"'}
	{attribute 'Tags' := '"LCID": "1033", "Text": "H, General, HtgCir, Operating mode"'}
	{attribute 'Description' := '"LCID": "1031", "Text": "Betriebsart"'}
	{attribute 'Description' := '"LCID": "1033", "Text": "Operating mode"'}
{endregion}
FUNCTION_BLOCK FB_BA_H_OpMod EXTENDS FB_BA_View
VAR_INPUT
	bDst					: BOOL;
	bHtgLmt					: BOOL;
	bTWthLowLimit			: BOOL;
END_VAR
VAR_OUTPUT
	eOpMod					: E_BA_EnergyLvl;
	bRls					: BOOL;
END_VAR
VAR_INPUT CONSTANT
	OpModMan				: FB_BA_MV_Op;
	Sched					: FB_BA_SchedM;
	OpModPr					: FB_BA_MV_Op;								 
	Rls						: FB_BA_BV_Op;
END_VAR
VAR
	OpModSwi				: FB_BA_PrioSwi_UDI08;
	RlsMMux					: FB_BA_MMUX_B04;
END_VAR

SUPER^(); // FB_BA_View
OpModMan(); // FB_BA_MV_Op
Sched(); // FB_BA_SchedM
OpModSwi(
    bEn01 := bDst,
    nVal01 := E_BA_EnergyLvl.eProtection,
    bEn02 := OpModMan.nPresentValue = E_BA_EnergyLvlA.eProtection,
    nVal02 := E_BA_EnergyLvl.eProtection,
    bEn03 := OpModMan.nPresentValue = E_BA_EnergyLvlA.eEconomy,
    nVal03 := E_BA_EnergyLvl.eEconomy,
    bEn04 := OpModMan.nPresentValue = E_BA_EnergyLvlA.eComfort,
    nVal04 := E_BA_EnergyLvl.eComfort,
    bEn05 := NOT bHtgLmt,
    nVal05 := E_BA_EnergyLvl.eProtection,
    bEn06 := Sched.nPresentValue = E_BA_EnergyLvl.eProtection,
    nVal06 := E_BA_EnergyLvl.eProtection,
    bEn07 := Sched.nPresentValue = E_BA_EnergyLvl.eEconomy,
    nVal07 := E_BA_EnergyLvl.eEconomy,
    bEn08 := Sched.nPresentValue = E_BA_EnergyLvl.eComfort,
    nVal08 := E_BA_EnergyLvl.eComfort); // FB_BA_PrioSwi_UDI08
OpModPr(nValuePgm := OpModSwi.nVal); // FB_BA_MV_Op
eOpMod := OpModPr.nPresentValue;
RlsMMux(
    bEn := TRUE,
    nSel := eOpMod,
    nEn01 := E_BA_EnergyLvl.eProtection,
    bVal01 := bTWthLowLimit,
    nEn02 := E_BA_EnergyLvl.eEconomy,
    bVal02 := TRUE,
    nEn03 := E_BA_EnergyLvl.eComfort,
    bVal03 := TRUE); // FB_BA_MMUX_B04
Rls(bValuePgm := RlsMMux.bVal); // FB_BA_BV_Op
bRls := Rls.bPresentValue;

METHOD FB_init : BOOL
VAR_INPUT
	bInitRetains : BOOL; // if TRUE, the retain variables are initialized (warm start / cold start)
	bInCopyCode : BOOL;  // if TRUE, the instance afterwards gets moved into the copy code (online change)
END_VAR
OpModMan.iParent		:= THIS^;
OpModMan.iLabel			:= LblCmpHeating.H_OpMod_OpModMan;							
OpModMan.sObjectName	:= '{Idx=01}';								 	 
OpModMan.aStateText[1]	:= txtEvent_Auto;
OpModMan.aStateText[2]	:= txtEvent_Protection;
OpModMan.aStateText[3]	:= txtEvent_Economy;
OpModMan.aStateText[4]	:= txtEvent_Comfort;
OpModMan.nValueRm		:= 1;

OpModPr.iParent			:= THIS^;
OpModPr.iLabel			:= LblCmpHeating.H_OpMod_OpModPr;							
OpModPr.sObjectName		:= '{Idx=01}';								 	 
OpModPr.aStateText[1]	:= txtEvent_Protection; 
OpModPr.aStateText[2]	:= txtEvent_Economy; 
OpModPr.aStateText[3]	:= txtEvent_Comfort; 
OpModPr.nValueRm		:= 1;

Rls.iParent				:= THIS^;
Rls.iLabel				:= LblCmpHeating.H_OpMod_Rls;	
Rls.sObjectName			:= '{Idx=01}';								 	 
Rls.sInactiveText		:= txtEvent_Off;
Rls.sActiveText			:= txtEvent_On;	
Rls.bValueRm			:= FALSE;								
Rls.eToggleMode 		:= E_BA_ToggleMode.eSwitch;	

Sched.iParent											:= THIS^;
Sched.iLabel											:= LblCmpHeating.H_OpMod_Sched;							
Sched.sObjectName										:= '{Idx=01}';								 	 
Sched.aStateText[1]										:= txtEvent_Protection;
Sched.aStateText[2]										:= txtEvent_Economy;
Sched.aStateText[3]										:= txtEvent_Comfort;
Sched.nPredictTime										:= 0;
Sched.nDefaultValue										:= E_BA_EnergyLvl.eProtection;
Sched.bWriteWeekly										:= FALSE;
//	Monday
Sched.aWeek[E_BA_Weekday.eMonday,1].eState				:= E_BA_SchedEntryState.eValue;
Sched.aWeek[E_BA_Weekday.eMonday,1].uValue.udiVal		:= E_BA_EnergyLvl.eComfort;
Sched.aWeek[E_BA_Weekday.eMonday,1].stTime.nHour		:= 6;
Sched.aWeek[E_BA_Weekday.eMonday,1].stTime.nMinute		:= 0;
Sched.aWeek[E_BA_Weekday.eMonday,1].stTime.nSecond		:= 0;
Sched.aWeek[E_BA_Weekday.eMonday,2].eState				:= E_BA_SchedEntryState.eValue;
Sched.aWeek[E_BA_Weekday.eMonday,2].uValue.udiVal		:= E_BA_EnergyLvl.eEconomy;
Sched.aWeek[E_BA_Weekday.eMonday,2].stTime.nHour		:= 20;
Sched.aWeek[E_BA_Weekday.eMonday,2].stTime.nMinute		:= 0;
Sched.aWeek[E_BA_Weekday.eMonday,2].stTime.nSecond		:= 0;
Sched.aWeek[E_BA_Weekday.eMonday,3].eState				:= E_BA_SchedEntryState.eValue;
Sched.aWeek[E_BA_Weekday.eMonday,3].uValue.udiVal		:= E_BA_EnergyLvl.eProtection;
Sched.aWeek[E_BA_Weekday.eMonday,3].stTime.nHour		:= 0;
Sched.aWeek[E_BA_Weekday.eMonday,3].stTime.nMinute		:= 0;
Sched.aWeek[E_BA_Weekday.eMonday,3].stTime.nSecond		:= 0;
//	Tuesday
Sched.aWeek[E_BA_Weekday.eTuesday,1].eState				:= E_BA_SchedEntryState.eValue;
Sched.aWeek[E_BA_Weekday.eTuesday,1].uValue.udiVal		:= E_BA_EnergyLvl.eComfort;
Sched.aWeek[E_BA_Weekday.eTuesday,1].stTime.nHour		:= 6;
Sched.aWeek[E_BA_Weekday.eTuesday,1].stTime.nMinute		:= 0;
Sched.aWeek[E_BA_Weekday.eTuesday,1].stTime.nSecond		:= 0;
Sched.aWeek[E_BA_Weekday.eTuesday,2].eState				:= E_BA_SchedEntryState.eValue;
Sched.aWeek[E_BA_Weekday.eTuesday,2].uValue.udiVal		:= E_BA_EnergyLvl.eEconomy;
Sched.aWeek[E_BA_Weekday.eTuesday,2].stTime.nHour		:= 20;
Sched.aWeek[E_BA_Weekday.eTuesday,2].stTime.nMinute		:= 0;
Sched.aWeek[E_BA_Weekday.eTuesday,2].stTime.nSecond		:= 0;
Sched.aWeek[E_BA_Weekday.eTuesday,3].eState				:= E_BA_SchedEntryState.eValue;
Sched.aWeek[E_BA_Weekday.eTuesday,3].uValue.udiVal		:= E_BA_EnergyLvl.eProtection;
Sched.aWeek[E_BA_Weekday.eTuesday,3].stTime.nHour		:= 0;
Sched.aWeek[E_BA_Weekday.eTuesday,3].stTime.nMinute		:= 0;
Sched.aWeek[E_BA_Weekday.eTuesday,3].stTime.nSecond		:= 0;
//	Wednesday
Sched.aWeek[E_BA_Weekday.eWednesday,1].eState			:= E_BA_SchedEntryState.eValue;
Sched.aWeek[E_BA_Weekday.eWednesday,1].uValue.udiVal	:= E_BA_EnergyLvl.eComfort;
Sched.aWeek[E_BA_Weekday.eWednesday,1].stTime.nHour		:= 6;
Sched.aWeek[E_BA_Weekday.eWednesday,1].stTime.nMinute	:= 0;
Sched.aWeek[E_BA_Weekday.eWednesday,1].stTime.nSecond	:= 0;
Sched.aWeek[E_BA_Weekday.eWednesday,2].eState			:= E_BA_SchedEntryState.eValue;
Sched.aWeek[E_BA_Weekday.eWednesday,2].uValue.udiVal	:= E_BA_EnergyLvl.eEconomy;
Sched.aWeek[E_BA_Weekday.eWednesday,2].stTime.nHour		:= 20;
Sched.aWeek[E_BA_Weekday.eWednesday,2].stTime.nMinute	:= 0;
Sched.aWeek[E_BA_Weekday.eWednesday,2].stTime.nSecond	:= 0;
Sched.aWeek[E_BA_Weekday.eWednesday,3].eState			:= E_BA_SchedEntryState.eValue;
Sched.aWeek[E_BA_Weekday.eWednesday,3].uValue.udiVal	:= E_BA_EnergyLvl.eProtection;
Sched.aWeek[E_BA_Weekday.eWednesday,3].stTime.nHour		:= 0;
Sched.aWeek[E_BA_Weekday.eWednesday,3].stTime.nMinute	:= 0;
Sched.aWeek[E_BA_Weekday.eWednesday,3].stTime.nSecond	:= 0;
//	Thursday
Sched.aWeek[E_BA_Weekday.eThursday,1].eState			:= E_BA_SchedEntryState.eValue;
Sched.aWeek[E_BA_Weekday.eThursday,1].uValue.udiVal		:=E_BA_EnergyLvl.eComfort;
Sched.aWeek[E_BA_Weekday.eThursday,1].stTime.nHour		:= 6;
Sched.aWeek[E_BA_Weekday.eThursday,1].stTime.nMinute	:= 0;
Sched.aWeek[E_BA_Weekday.eThursday,1].stTime.nSecond	:= 0;
Sched.aWeek[E_BA_Weekday.eThursday,2].eState			:= E_BA_SchedEntryState.eValue;
Sched.aWeek[E_BA_Weekday.eThursday,2].uValue.udiVal		:= E_BA_EnergyLvl.eEconomy;
Sched.aWeek[E_BA_Weekday.eThursday,2].stTime.nHour		:= 20;
Sched.aWeek[E_BA_Weekday.eThursday,2].stTime.nMinute	:= 0;
Sched.aWeek[E_BA_Weekday.eThursday,2].stTime.nSecond	:= 0;
Sched.aWeek[E_BA_Weekday.eThursday,3].eState			:= E_BA_SchedEntryState.eValue;
Sched.aWeek[E_BA_Weekday.eThursday,3].uValue.udiVal		:= E_BA_EnergyLvl.eProtection;
Sched.aWeek[E_BA_Weekday.eThursday,3].stTime.nHour		:= 0;
Sched.aWeek[E_BA_Weekday.eThursday,3].stTime.nMinute	:= 0;
Sched.aWeek[E_BA_Weekday.eThursday,3].stTime.nSecond	:= 0;
//	Friday
Sched.aWeek[E_BA_Weekday.eFriday,1].eState				:= E_BA_SchedEntryState.eValue;
Sched.aWeek[E_BA_Weekday.eFriday,1].uValue.udiVal		:= E_BA_EnergyLvl.eComfort;
Sched.aWeek[E_BA_Weekday.eFriday,1].stTime.nHour		:= 6;
Sched.aWeek[E_BA_Weekday.eFriday,1].stTime.nMinute		:= 0;
Sched.aWeek[E_BA_Weekday.eFriday,1].stTime.nSecond		:= 0;
Sched.aWeek[E_BA_Weekday.eFriday,2].eState				:= E_BA_SchedEntryState.eValue;
Sched.aWeek[E_BA_Weekday.eFriday,2].uValue.udiVal		:= E_BA_EnergyLvl.eEconomy;
Sched.aWeek[E_BA_Weekday.eFriday,2].stTime.nHour		:= 20;
Sched.aWeek[E_BA_Weekday.eFriday,2].stTime.nMinute		:= 0;
Sched.aWeek[E_BA_Weekday.eFriday,2].stTime.nSecond		:= 0;
Sched.aWeek[E_BA_Weekday.eFriday,3].eState				:= E_BA_SchedEntryState.eValue;
Sched.aWeek[E_BA_Weekday.eFriday,3].uValue.udiVal		:= E_BA_EnergyLvl.eProtection;
Sched.aWeek[E_BA_Weekday.eFriday,3].stTime.nHour		:= 0;
Sched.aWeek[E_BA_Weekday.eFriday,3].stTime.nMinute		:= 0;
Sched.aWeek[E_BA_Weekday.eFriday,3].stTime.nSecond		:= 0;
END_METHOD

END_FUNCTION_BLOCK

// ---- Templates/POUs/Trade/HeatingSystem/Setpoint/FB_BA_H_HtgCir_Sp.TcPOU
{region '#Template'}
	{attribute 'Version' := '1.0.0.0'}
	{attribute 'Tags' := '"LCID": "1031", "Text": "H, Heating circuit, HtgCir, Setpoint"'}
	{attribute 'Tags' := '"LCID": "1033", "Text": "H, Heating circuit, HtgCir, Setpoint"'}
	{attribute 'Description' := '"LCID": "1031", "Text": "Sollwert Heizkreis"'}
	{attribute 'Description' := '"LCID": "1033", "Text": "Setpoint heating circuit"'}
{endregion}
FUNCTION_BLOCK FB_BA_H_HtgCir_Sp EXTENDS FB_BA_View
VAR_INPUT
	eOpMod					: E_BA_EnergyLvl;
	fSpFrstProtec			: REAL;
	fTWthDamp				: REAL;
END_VAR
VAR_OUTPUT
	fSpFlWT							: REAL;
END_VAR
VAR_INPUT CONSTANT
	NgtOffs					: FB_BA_AV_Op;	
	SpFlWT					: FB_BA_AV_Op;		
	HtgCrv					: FB_BA_Scale_04; 
END_VAR
VAR
	PrioSwi					: FB_BA_MMUX_R04;
END_VAR

// note: 1 stored wires end on pins the file does not list and are not shown
SUPER^(); // FB_BA_View
NgtOffs(); // FB_BA_AV_Op
HtgCrv(fX := fTWthDamp); // FB_BA_Scale_04
PrioSwi(
    bEn := TRUE,
    nSel := eOpMod,
    nEn01 := E_BA_EnergyLvl.eComfort,
    fVal01 := HtgCrv.fY,
    nEn02 := E_BA_EnergyLvl.eEconomy,
    fVal02 := HtgCrv.fY - ABS(NgtOffs.fPresentValue),
    nEn03 := E_BA_EnergyLvl.eProtection,
    fVal03 := fSpFrstProtec); // FB_BA_MMUX_R04
SpFlWT(fValuePgm := PrioSwi.fVal); // FB_BA_AV_Op
fSpFlWT := SpFlWT.fPresentValue;

METHOD FB_init : BOOL
VAR_INPUT
	bInitRetains : BOOL; // if TRUE, the retain variables are initialized (warm start / cold start)
	bInCopyCode : BOOL;  // if TRUE, the instance afterwards gets moved into the copy code (online change)
END_VAR
NgtOffs.iParent				:= THIS^;
NgtOffs.iLabel				:= LblCmpHeating.H_HtgCir_Sp_NgtOffs;		 
NgtOffs.sObjectName			:= '{Idx=01}';
NgtOffs.eUnit				:= E_BA_Unit.eTemperature_DegreesCelsius;  
NgtOffs.fValueRm			:= 8.0;
NgtOffs.fCOVIncrement	:= BA2_Param.fDefCOVIncrement;							

SpFlWT.iParent				:= THIS^;
SpFlWT.iLabel				:= LblCmpHeating.H_HtgCir_Sp_SpFlWT;		 
SpFlWT.sObjectName			:= '{Idx=01}';
SpFlWT.eUnit				:= E_BA_Unit.eTemperature_DegreesCelsius;  
SpFlWT.fCOVIncrement		:= BA2_Param.fDefCOVIncrement;							

HtgCrv.iParent				:= THIS^;										
HtgCrv.iLabel				:= LblCmpHeating.H_HtgCir_Sp_HtgCrv;
HtgCrv.sObjectName			:= '{Idx=01}';										 
HtgCrv.eDPADMode			:= E_BA_DPADMode.eIncludeDescription; 
HtgCrv.X1.fValueRm			:= 15.0;
HtgCrv.X2.fValueRm			:= 0.0;
HtgCrv.X3.fValueRm			:= -10.0;
HtgCrv.X4.fValueRm			:= -20.0;
HtgCrv.Y1.fValueRm			:= 25.0;
HtgCrv.Y2.fValueRm			:= 40.0;
HtgCrv.Y3.fValueRm			:= 55.0;
HtgCrv.Y4.fValueRm			:= 65.0;
HtgCrv.YMin.fValueRm		:= 5.0;
HtgCrv.YMax.fValueRm		:= 80.0;
END_METHOD

END_FUNCTION_BLOCK

// ---- Templates/POUs/Universal/Aggregat/Binary/FB_BA_ActuatorCmd.TcPOU
{region '#Template'}
	{attribute 'Version' := '0.0.1.0'}
	{attribute 'Tags' := '"LCID": "1031", "Text": "Universal, Analog, Aggregate"'}
	{attribute 'Tags' := '"LCID": "1033", "Text": "Universal, Analog, Aggregate"'}
	{attribute 'Description' := '"LCID": "1031", "Text": "Aktor binär"'}
	{attribute 'Description' := '"LCID": "1033", "Text": "Actuator binary"'}
{endregion}
FUNCTION_BLOCK FB_BA_ActuatorCmd EXTENDS FB_BA_AggregateB
VAR_OUTPUT
	bCmd							: BOOL;
END_VAR
VAR_INPUT CONSTANT
	Cmd						: FB_BA_BO_IO;			
END_VAR

SUPER^(); // FB_BA_AggregateB
Cmd(
    bEnSfty := bEnSfty,
    bValSfty := SUPER^.bActiveVal,
    bEnCrit := bEnCrit,
    bValCrit := SUPER^.bActiveVal,
    bEnPgm := bEnPgm,
    bValPgm := SUPER^.bActiveVal); // FB_BA_BO_IO
bCmd := Cmd.bPresentValue;

